    // =========================================================================
    // [1] RegisterAlarm ID — 倉儲區氣缸 (500-599) [Hold, Level2]
    // =========================================================================
    GC_ALARM_CYL_STO_UPCV_FEEDIN1       : DINT := 500;   // 上CV進料壓缸1
    GC_ALARM_CYL_STO_UPCV_FEEDIN2       : DINT := 501;   // 上CV進料壓缸2
    GC_ALARM_CYL_STO_UPCV_DIAMETER      : DINT := 502;   // 上CV量徑壓缸
    GC_ALARM_CYL_STO_UPCV_CAM1          : DINT := 503;   // 上CV相機壓缸1
    GC_ALARM_CYL_STO_UPCV_CAM2          : DINT := 504;   // 上CV相機壓缸2
    GC_ALARM_CYL_STO_UPCV_CAM3          : DINT := 505;   // 上CV相機壓缸3
    GC_ALARM_CYL_STO_UPCV_CAM4          : DINT := 506;   // 上CV相機壓缸4
    GC_ALARM_CYL_STO_UPCV_BLOCK1        : DINT := 507;   // 上CV擋塊1
    GC_ALARM_CYL_STO_UPCV_BLOCK2        : DINT := 508;   // 上CV擋塊2
    GC_ALARM_CYL_STO_UPCV_BLOCK3        : DINT := 509;   // 上CV擋塊3
    GC_ALARM_CYL_STO_UPCV_DIA_HORIZ     : DINT := 510;   // 上CV量徑水平
    GC_ALARM_CYL_STO_UPCV_DIA_VERT      : DINT := 511;   // 上CV量徑垂直
    GC_ALARM_CYL_STO_UPCV_DIA_CLAMP     : DINT := 512;   // 上CV量徑夾
    GC_ALARM_CYL_STO_STACK_PUSH         : DINT := 513;   // 疊盒推缸
    GC_ALARM_CYL_STO_LOWCV_PRESS1       : DINT := 514;   // 下CV壓缸1
    GC_ALARM_CYL_STO_LOWCV_PRESS2       : DINT := 515;   // 下CV壓缸2
    GC_ALARM_CYL_STO_LOWCV_PRESS3       : DINT := 516;   // 下CV壓缸3
    GC_ALARM_CYL_STO_LOWCV_PRESS4       : DINT := 517;   // 下CV壓缸4
    GC_ALARM_CYL_STO_LOWCV_BLOCK1       : DINT := 518;   // 下CV擋塊1
    GC_ALARM_CYL_STO_LOWCV_BLOCK2       : DINT := 519;   // 下CV擋塊2
    GC_ALARM_CYL_STO_SAME_BLOCK3        : DINT := 520;   // 同徑CV擋塊3
    GC_ALARM_CYL_STO_SHIP_BUFFER        : DINT := 521;   // 出貨緩衝壓缸
    // 522-599: 預留倉儲區氣缸擴充

    // =========================================================================
    // [1] RegisterAlarm ID — 配針區氣缸 (600-699) [Hold, Level2]
    // =========================================================================
    GC_ALARM_CYL_ALC_ROBOT_LCLAMP1      : DINT := 600;   // AllocateRobot 左夾1
    GC_ALARM_CYL_ALC_ROBOT_LCLAMP2      : DINT := 601;   // AllocateRobot 左夾2
    GC_ALARM_CYL_ALC_ROBOT_LVERT1       : DINT := 602;   // AllocateRobot 左升降1
    GC_ALARM_CYL_ALC_ROBOT_LVERT2       : DINT := 603;   // AllocateRobot 左升降2
    GC_ALARM_CYL_ALC_ROBOT_RCLAMP1      : DINT := 604;   // AllocateRobot 右夾1
    GC_ALARM_CYL_ALC_ROBOT_RCLAMP2      : DINT := 605;   // AllocateRobot 右夾2
    GC_ALARM_CYL_ALC_ROBOT_RVERT1       : DINT := 606;   // AllocateRobot 右升降1
    GC_ALARM_CYL_ALC_ROBOT_RVERT2       : DINT := 607;   // AllocateRobot 右升降2
    GC_ALARM_CYL_ALC_DIFF_BLOCK1        : DINT := 608;   // 異徑CV擋塊1
    GC_ALARM_CYL_ALC_RB_WORK_PRESS      : DINT := 609;   // 圓帶工作區壓缸
    GC_ALARM_CYL_ALC_RB_WORK_PLUG       : DINT := 610;   // 圓帶工作區插銷
    GC_ALARM_CYL_ALC_RB_CHARGE_PLUG     : DINT := 611;   // 圓帶充電區插銷
    GC_ALARM_CYL_ALC_RB_TRANS_PLUG      : DINT := 612;   // 圓帶傳送區插銷
    GC_ALARM_CYL_ALC_OUTROBOT_AVERT     : DINT := 613;   // OutRobot A側升降
    GC_ALARM_CYL_ALC_OUTROBOT_BVERT     : DINT := 614;   // OutRobot B側升降
    GC_ALARM_CYL_ALC_OUTROBOT_ACLAMP    : DINT := 615;   // OutRobot A側夾
    GC_ALARM_CYL_ALC_OUTROBOT_BCLAMP    : DINT := 616;   // OutRobot B側夾
    GC_ALARM_CYL_ALC_TRANS_CAMHORIZ     : DINT := 617;   // 傳送CV相機水平
    GC_ALARM_CYL_ALC_DIFF_PRESS2        : DINT := 618;   // 異徑CV壓缸2
    GC_ALARM_CYL_ALC_DIFF_PRESS1        : DINT := 619;   // 異徑CV壓缸1
    GC_ALARM_CYL_ALC_DIFF_BLOCK1_2      : DINT := 620;   // 異徑CV擋塊1 (重複)
    GC_ALARM_CYL_ALC_SAME_PRESS4        : DINT := 621;   // 同徑CV壓缸4
    GC_ALARM_CYL_ALC_SAME_PRESS3        : DINT := 622;   // 同徑CV壓缸3
    GC_ALARM_CYL_ALC_SAME_PRESS2        : DINT := 623;   // 同徑CV壓缸2
    GC_ALARM_CYL_ALC_SAME_PRESS1        : DINT := 624;   // 同徑CV壓缸1
    GC_ALARM_CYL_ALC_SAME_BLOCK2        : DINT := 625;   // 同徑CV擋塊2
    GC_ALARM_CYL_ALC_SAME_BLOCK1        : DINT := 626;   // 同徑CV擋塊1
    GC_ALARM_CYL_ALC_PULLOUT_APRESS1    : DINT := 627;   // 拔針CV A側壓缸1
    GC_ALARM_CYL_ALC_PULLOUT_APRESS2    : DINT := 628;   // 拔針CV A側壓缸2
    GC_ALARM_CYL_ALC_PULLOUT_ABLOCK     : DINT := 629;   // 拔針CV A側擋塊
    GC_ALARM_CYL_ALC_PULLOUT_BPRESS1    : DINT := 630;   // 拔針CV B側壓缸1
    GC_ALARM_CYL_ALC_PULLOUT_BPRESS2    : DINT := 631;   // 拔針CV B側壓缸2
    GC_ALARM_CYL_ALC_PULLOUT_BBLOCK     : DINT := 632;   // 拔針CV B側擋塊
    // 633-699: 預留配針區氣缸擴充

    // =========================================================================
    // [1] RegisterAlarm ID — 伺服軸 (800-899) [Abort, Level6]
    // =========================================================================
    GC_ALARM_AXIS_TURNTABLE              : DINT := 800;   // [Abort] 轉盤軸錯誤
    GC_ALARM_AXIS_ROUNDBELT              : DINT := 801;   // [Abort] 圓帶軸錯誤
    GC_ALARM_AXIS_ALLOCATE_X             : DINT := 802;   // [Abort] 配針X軸錯誤
    GC_ALARM_AXIS_ALLOCATE_Y             : DINT := 803;   // [Abort] 配針Y軸錯誤
    GC_ALARM_AXIS_OUTROBOT_X             : DINT := 804;   // [Abort] OutRobot X軸錯誤
    GC_ALARM_AXIS_OUTROBOT_Y             : DINT := 805;   // [Abort] OutRobot Y軸錯誤
    GC_ALARM_AXIS_RACKMOTOR              : DINT := 806;   // [Abort] RackMotor軸錯誤
    // 807-899: 預留伺服軸擴充
	
	GC_ALARM_MODBUSRTU					: DINT	:= 850;	  // 光電板 MODBUS (實際用 +1 ~ +4) 

    // =========================================================================
    // [1] RegisterAlarm ID — 安全門 (900-999) [Hold, Level2]
    // =========================================================================
    GC_ALARM_SAFE_DOOR_BASE              : DINT := 900;   // 安全門基底 (實際用 +1 ~ +16)
    // 917-999: 預留安全相關擴充

    // =========================================================================
    // [2] FB 內部錯誤碼 — 通用 (A=0, OO=00 一般)
    // =========================================================================
    GC_ERR_NONE                          : INT := 0;       // 無錯誤
    GC_ERR_TIMEOUT                       : INT := 1;       // 逾時 [Hold]
    GC_ERR_POSITION_INVALID              : INT := 3;       // 位置資料無效 [Hold]
    GC_ERR_INDEX_INVALID                 : INT := 10;      // 索引無效 [Hold]
    GC_ERR_WRONG_COMMAND                 : INT := 11;      // 錯誤指令 [Hold]
    GC_ERR_ROBOT_NUMBER_INVALID          : INT := 12;      // 機器人編號無效 [Hold]

    // -- 通用 氣缸 (A=0, OO=01) --
    GC_ERR_CYLINDER_NOT_READY            : INT := 102;     // 氣缸未就緒 [Hold]

    // -- 通用 馬達 (A=0, OO=02) --
    GC_ERR_MOTOR_NOT_READY               : INT := 202;     // 馬達未就緒 [Hold]

    // -- 通用 伺服軸 (A=0, OO=03) --
    GC_ERR_AXIS_NOT_READY                : INT := 302;     // 軸未就緒 [Hold]
    GC_ERR_AXIS_ERROR                    : INT := 310;     // 軸錯誤 [Abort]
    GC_ERR_AXIS_POSITION_ERROR           : INT := 305;     // 軸位置錯誤 [Hold]
    GC_ERR_AXIS_SAFETY_CALL_ERROR        : INT := 311;     // 呼叫軸安全檢查錯誤 [Abort]
    GC_ERR_AXIS_SAFETY_CHECK_ERROR       : INT := 312;     // 軸安全檢查錯誤 [Abort]
    GC_ERR_AXIS_OUTROBOT_X_ERROR        : INT := 313;     // OutRobot X軸錯誤 [Abort]
    GC_ERR_AXIS_OUTROBOT_Y_ERROR        : INT := 314;     // OutRobot Y軸錯誤 [Abort]
    GC_ERR_AXIS_ALLOCATE_X_ERROR        : INT := 315;     // 配針X軸錯誤 [Abort]
    GC_ERR_AXIS_ALLOCATE_Y_ERROR        : INT := 316;     // 配針Y軸錯誤 [Abort]
    GC_ERR_AXIS_ROUNDBELT_ERROR         : INT := 317;     // 圓帶軸錯誤 [Abort]
    GC_ERR_AXIS_TURNTABLE_ERROR         : INT := 318;     // 轉盤軸錯誤 [Abort]
    GC_ERR_RACKMOTOR_BTN_BLINK          : INT := 319;     // RackMotor按鈕閃爍 [Hold]
    GC_ERR_AXIS_X_NOT_READY             : INT := 320;     // X軸未就緒 [Hold]
    GC_ERR_AXIS_Y_NOT_READY             : INT := 321;     // Y軸未就緒 [Hold]

    // -- 通用 機器人 (A=0, OO=04) --
    GC_ERR_ROBOT_CANNOT_HOME             : INT := 410;     // 機器人無法回原點 [Abort]
    GC_ERR_ROBOT_REBOOT_TIMEOUT          : INT := 411;     // 機器人重啟逾時 [Abort]
    GC_ERR_ROBOT_CMD_NOT_BUSY            : INT := 412;     // 機器人指令未接受 [Hold]
    GC_ERR_ROBOT_CMD_TIMEOUT             : INT := 413;     // 機器人指令完成逾時 [Abort]
    GC_ERR_ROBOT_HOMING_ERROR            : INT := 414;     // 機器人回原點錯誤+訊息 [Abort]

    // =========================================================================
    // [2] FB 內部錯誤碼 — 倉儲區專用 (A=1)
    // =========================================================================
    GC_ERR_STO_ROBOT_FEEDOUT_NOT_BUSY    : INT := 10412;   // 倉儲機器人 FeedOut 未接受 [Hold]
    GC_ERR_STO_ROBOT_FEEDOUT_TIMEOUT     : INT := 10413;   // 倉儲機器人 FeedOut 逾時 [Abort]
    GC_ERR_STO_SERVICE_OCCUPIED          : INT := 10006;   // 倉儲服務佔用中 [Hold]

    // -- 倉儲區 下CV輸送帶 (A=1, OO=05/01) --
    GC_ERR_STO_LOWCV_BLOCK1_ERROR       : INT := 10110;   // 下CV擋塊1錯誤 [Hold]
    GC_ERR_STO_LOWCV_BLOCK2_ERROR       : INT := 10111;   // 下CV擋塊2錯誤 [Hold]
    GC_ERR_STO_LOWCV_PRESS1_ERROR       : INT := 10112;   // 下CV壓缸1錯誤 [Hold]
    GC_ERR_STO_LOWCV_PRESS2_ERROR       : INT := 10113;   // 下CV壓缸2錯誤 [Hold]
    GC_ERR_STO_LOWCV_PRESS3_ERROR       : INT := 10114;   // 下CV壓缸3錯誤 [Hold]
    GC_ERR_STO_LOWCV_PRESS4_ERROR       : INT := 10115;   // 下CV壓缸4錯誤 [Hold]
    GC_ERR_STO_LOWCV_BOX_TIMEOUT        : INT := 10501;   // 下CV盒子到位逾時 [Hold]
    GC_ERR_STO_LOWCV_CYL_ERROR          : INT := 10116;   // 下CV氣缸錯誤 (CyclicAction) [Hold]
    GC_ERR_STO_LOWCV_MOTOR_ERROR        : INT := 10201;   // 下CV馬達錯誤 (CyclicAction) [Hold]

    // =========================================================================
    // [2] FB 內部錯誤碼 — 配針區專用 (A=2)
    // =========================================================================
    GC_ERR_ALC_RB_NOT_READY              : INT := 20602;   // 圓帶軸未就緒 [Hold]
    GC_ERR_ALC_RB_CYLINDER_ERROR         : INT := 20102;   // 圓帶氣缸錯誤 [Hold]
    GC_ERR_ALC_RB_AXIS_ERROR             : INT := 20610;   // 圓帶軸錯誤 [Abort]
    GC_ERR_ALC_RB_CHARGE_PLUG_ERROR      : INT := 20111;   // 充電區插銷錯誤 [Hold]
    GC_ERR_ALC_RB_TRANSMITCV_PLUG_ERROR  : INT := 20511;   // 傳送帶插銷錯誤 [Hold]
    GC_ERR_ALC_RB_WORKZONE_PLUG_ERROR    : INT := 20112;   // 工作區插銷錯誤 [Hold]
    GC_ERR_ALC_RB_WORKZONE_PRESS_ERROR   : INT := 20113;   // 工作區壓缸錯誤 [Hold]
    GC_ERR_ALC_SERVO_ERROR               : INT := 20310;   // 配針伺服軸錯誤 [Abort]

    // -- 配針區 轉盤 (A=2, OO=07) --
    GC_ERR_ALC_TT_TARGET_INVALID        : INT := 20703;   // 轉盤目標無效 [Hold]
    GC_ERR_ALC_TT_AXIS_NOT_READY        : INT := 20702;   // 轉盤軸未就緒 [Hold]
    GC_ERR_ALC_TT_AXIS_ERROR            : INT := 20710;   // 轉盤軸錯誤 [Abort]
    GC_ERR_ALC_TT_CYLINDER_NOT_READY    : INT := 20701;   // 轉盤氣缸未就緒 [Hold]
    GC_ERR_ALC_TT_PRESS_ERROR           : INT := 20711;   // 轉盤壓缸錯誤 [Hold]

    // -- 配針區 同徑CV相機 (A=2) --
    GC_ERR_ALC_SAMECV_BLOCK1_ERROR      : INT := 20120;   // 同徑CV Block1錯誤 [Hold]
    GC_ERR_ALC_SAMECV_BLOCK2_ERROR      : INT := 20121;   // 同徑CV Block2錯誤 [Hold]
    GC_ERR_ALC_SAMECV_PRESS1_ERROR      : INT := 20122;   // 同徑CV Press1錯誤 [Hold]
    GC_ERR_ALC_SAMECV_PRESS2_ERROR      : INT := 20123;   // 同徑CV Press2錯誤 [Hold]
    GC_ERR_ALC_SAMECV_CAMHORIZ_ERROR    : INT := 20124;   // 同徑CV CameraHoriz錯誤 [Hold]
    GC_ERR_ALC_SAMECV_BOX_NOT_ARRIVED   : INT := 20515;   // 同徑CV 盒子未到逾時 [Hold]
    GC_ERR_ALC_SAMECV_CYL_TIMEOUT       : INT := 20125;   // 同徑CV 氣缸逾時 [Hold]
    GC_ERR_ALC_SAMECV_CAMERA_TIMEOUT    : INT := 20516;   // 同徑CV 拍照逾時 [Abort]
    GC_ERR_ALC_SAMECV_BOX_CROSS_TIMEOUT : INT := 20517;   // 同徑CV 盒子通過逾時 [Hold]
    GC_ERR_ALC_SAMECV_FULL              : INT := 20518;   // 同徑CV 滿載 [Hold]
    GC_ERR_ALC_SAMECV_MOTOR_ERROR       : INT := 20225;   // 同徑CV 馬達錯誤 [Hold]

    // -- 配針區 異徑CV相機 (A=2) --
    GC_ERR_ALC_DIFFCV_BLOCK1_ERROR      : INT := 20130;   // 異徑CV Block1錯誤 [Hold]
    GC_ERR_ALC_DIFFCV_PRESS1_ERROR      : INT := 20131;   // 異徑CV Press1錯誤 [Hold]
    GC_ERR_ALC_DIFFCV_CAMHORIZ_ERROR    : INT := 20132;   // 異徑CV CamaraHoriz錯誤 [Hold]
    GC_ERR_ALC_DIFFCV_NOT_READY         : INT := 20519;   // 異徑CV 未就緒 [Hold]
    GC_ERR_ALC_DIFFCV_CYL_TIMEOUT       : INT := 20133;   // 異徑CV 氣缸逾時 [Hold]
    GC_ERR_ALC_DIFFCV_BOX_NOT_ARRIVED   : INT := 20520;   // 異徑CV 盒子未到逾時 [Hold]
    GC_ERR_ALC_DIFFCV_CYL_MOTOR_TIMEOUT : INT := 20134;   // 異徑CV 馬達/氣缸逾時 [Hold]
    GC_ERR_ALC_DIFFCV_CAMERA_TIMEOUT    : INT := 20521;   // 異徑CV 拍照逾時 [Abort]
    GC_ERR_ALC_DIFFCV_BOX_CROSS_TIMEOUT : INT := 20522;   // 異徑CV 盒子通過逾時 [Hold]
    GC_ERR_ALC_DIFFCV_FULL              : INT := 20523;   // 異徑CV 滿載 [Hold]
    GC_ERR_ALC_DIFFCV_MOTOR_ERROR       : INT := 20226;   // 異徑CV 馬達錯誤 [Hold]

    // -- 配針區 逆向拍照批次入料 (A=2) --
    GC_ERR_ALC_REVBATCH_PICKUP_TIMEOUT  : INT := 20530;   // 逆向批次 小手臂取放盒逾時 [Hold]
    GC_ERR_ALC_REVBATCH_BIGARM_TIMEOUT  : INT := 20531;   // 逆向批次 大手臂搬運逾時 [Hold]
    GC_ERR_ALC_REVBATCH_CONVEYOR_FULL   : INT := 20532;   // 逆向批次 軌道滿載 [Hold]
    GC_ERR_ALC_REVBATCH_CONFIG_TIMEOUT  : INT := 20533;   // 逆向批次 等待C#配置逾時 [Hold]
    GC_ERR_ALC_REVBATCH_CAMERA_TIMEOUT  : INT := 20534;   // 逆向批次 拍照逾時 [Hold]

    // =========================================================================
    // [2] FB 內部錯誤碼 — 出貨區專用 (A=3)
    // =========================================================================
    GC_ERR_SHP_ROBOT_FEEDOUT_NOT_BUSY    : INT := 30412;   // 出貨機器人 FeedOut 未接受 [Hold]
    GC_ERR_SHP_ROBOT_FEEDOUT_TIMEOUT     : INT := 30413;   // 出貨機器人 FeedOut 逾時 [Abort]
    GC_ERR_SHP_SERVICE_OCCUPIED          : INT := 30006;   // 出貨服務佔用中 [Hold]
    GC_ERR_SHP_ROBOT_REBOOT_TIMEOUT      : INT := 30411;   // 出貨機器人重啟逾時 [Abort]

    // -- 出貨區 雷射/傳送帶 (A=3) --
    GC_ERR_SHP_LASER_ERROR              : INT := 30910;   // 雷射機台錯誤 [Hold]
    GC_ERR_SHP_TRANSCV_NOT_IN_POS       : INT := 30511;   // 傳送帶未在目標位置 [Hold]

    // =========================================================================
    // [3] 服務唯一識別碼 — UniqueErrorCode (INT)
    //     各 Service FB 的 ErrorID，用於錯誤追蹤定位
    // =========================================================================
    // -- 倉儲區機器人服務 --
    GC_SVCID_STO_ROBOT_ABS_MOVE         : INT := 2200;   // 倉儲機器人絕對移動
    GC_SVCID_STO_REGION_ALLOC_CV        : INT := 2210;   // 區域移動-配針輸送帶
    GC_SVCID_STO_REGION_ROUNDBELT       : INT := 2220;   // 區域移動-圓帶
    GC_SVCID_STO_REGION_PULLOUT_CV      : INT := 2230;   // 區域移動-拔針輸送帶
    GC_SVCID_STO_REGION_FEEDIN_CV       : INT := 2240;   // 區域移動-進料輸送帶
    GC_SVCID_STO_WAREHOUSE_ROBOT        : INT := 2400;   // 倉儲機器人移動
    GC_SVCID_STO_ADD_BOXES              : INT := 2700;   // 加盒服務
    GC_SVCID_STO_UPPER_FEEDIN_CV        : INT := 2710;   // 上層進料輸送帶
    GC_SVCID_STO_BOX_SUPPLY             : INT := 2800;   // 供盒控制

    // -- 配針區服務 --
    GC_SVCID_ALC_PULLOUT_CV             : INT := 2750;   // 拔針輸送帶
    GC_SVCID_ALC_BATCH_SIMPLE           : INT := 112;    // 批次配針(簡易模式)
    GC_SVCID_ALC_BATCH_FULL             : INT := 108;    // 批次配針(完整模式)

    // -- 出貨區機器人服務 --
    GC_SVCID_SHP_ROBOT                  : INT := 2250;   // 出貨機器人


    // =========================================================================
    // [3] 中央化狀態訊息常數
    // =========================================================================
    GC_MSG_0001                      : STRING := 'Action Robot timeout';
    GC_MSG_0002: STRING := 'BlockBox1 MoveForward or BlockBox2 MoveBackward or DiameterMeasurementPressBox MoveBackward timeout';
    GC_MSG_0003           : STRING := 'Block 1 cylinder inrearPosition';
    GC_MSG_0004           : STRING := 'Block 2 cylinder inrearPosition';
    GC_MSG_0005             : STRING := 'Block box on conveyor timeout';
    GC_MSG_0006                     : STRING := 'box1 diameter timeout';
    GC_MSG_0007: STRING := 'Box not at Input.bUpCV_Block2Detect_Sensor';
    GC_MSG_0008                      : STRING := 'Box not On Turntable';
    GC_MSG_0009                      : STRING := 'Box Not on Turntable';
    GC_MSG_0010                                 : STRING := 'Box on A1';
    GC_MSG_0011                                 : STRING := 'Box on A2';
    GC_MSG_0012                          : STRING := 'Box On Turntable';
    GC_MSG_0013                           : STRING := 'Box still on A1';
    GC_MSG_0014                           : STRING := 'Box still on A2';
    GC_MSG_0015                     : STRING := 'Box still on conveyor';
    GC_MSG_0016                    : STRING := 'Box still on Turntable';
    GC_MSG_0017       : STRING := 'Check FirstBoxCamaraDone info retry';
    GC_MSG_0018                        : STRING := 'ClampA Robot Error';
    GC_MSG_0019                    : STRING := 'Clamp A Feedin timeout';
    GC_MSG_0020                    : STRING := 'Clamp A reload timeout';
    GC_MSG_0021                     : STRING := 'Clamp A robot timeout';
    GC_MSG_0022                    : STRING := 'Clamp B Feedin timeout';
    GC_MSG_0023                    : STRING := 'Clamp B reload timeout';
    GC_MSG_0024                     : STRING := 'Clamp B Robot timeout';
    GC_MSG_0025                   : STRING := 'Clip pick close timeout';
    GC_MSG_0026                   : STRING := 'clip pick close timeout';
    GC_MSG_0027                   : STRING := 'clip place open timeout';
    GC_MSG_0028                   : STRING := 'Clip place open timeout';
    GC_MSG_0029: STRING := 'Command error : Clamp A target layer out of range.';
    GC_MSG_0030: STRING := 'Command error : Clamp A target slide out of range';
    GC_MSG_0031: STRING := 'Command error : Clamp B target layer out of range.';
    GC_MSG_0032: STRING := 'Command error : Clamp B target slide out of range';
    GC_MSG_0033                   : STRING := 'Controller report error';
    GC_MSG_0034: STRING := 'Conveyor not ready , please remove boxes in front';
    GC_MSG_0035: STRING := 'Cylinder.List.fbUpCV_Block2 MoveForward timeout';
    GC_MSG_0036       : STRING := 'Cylinder.List.fbUpCV_Block3 timeout';
    GC_MSG_0037: STRING := 'Cylinder.List.fbUpCV_CamaraPress1.M_MoveForward timeout';
    GC_MSG_0038: STRING := 'Cylinder.List.fbUpCV_CamaraPress1 or Cylinder.List.fbUpCV_Block3 InRearPosition timeout';
    GC_MSG_0039: STRING := 'Cylinder.List.fbUpCV_DiameterClamp M_Extend Timeout';
    GC_MSG_0040: STRING := 'Cylinder.List.fbUpCV_DiameterClamp M_Retract Timeout';
    GC_MSG_0041: STRING := 'Cylinder.List.fbUpCV_DiameterHoriz M_Extend Timeout';
    GC_MSG_0042: STRING := 'Cylinder.List.fbUpCV_DiameterHoriz M_Retract Timeout';
    GC_MSG_0043: STRING := 'Cylinder.List.fbUpCV_DiameterPress MoveForward timeout';
    GC_MSG_0044: STRING := 'Cylinder.List.fbUpCV_DiameterVert MoveForward Timeout';
    GC_MSG_0045: STRING := 'Cylinder.List.fbUpCV_DiameterVert M_Extend Timeout';
    GC_MSG_0046: STRING := 'Cylinder.List.fbUpCV_DiameterVert M_Retract Timeout';
    GC_MSG_0047: STRING := 'Cylinder.List.fbUpCV_FeedInPress1 or Cylinder.List.fbUpCV_FeedInPress2 MoveForward timeout';
    GC_MSG_0048                : STRING := 'Cylinder pick down timeout';
    GC_MSG_0049                  : STRING := 'Cylinder pick up timeout';
    GC_MSG_0050                  : STRING := 'cylinder pick up timeout';
    GC_MSG_0051               : STRING := 'Cylinder place down timeout';
    GC_MSG_0052                 : STRING := 'Cylinder place up timeout';
    GC_MSG_0053                 : STRING := 'cylinder place up timeout';
    GC_MSG_0054       : STRING := 'C# DiameterMovement Pickdone timeout';
    GC_MSG_0055   : STRING := 'C# FirstBoxCameraDiameterRequest timeout';
    GC_MSG_0056              : STRING := 'C# FirstBoxCameraDone timeout';
    GC_MSG_0057     : STRING := 'C# SecondBoxCameraDiameterDone timeout';
    GC_MSG_0058                          : STRING := 'Data not correct';
    GC_MSG_0059  : STRING := 'Destination: Left TransCV not in position';
    GC_MSG_0060 : STRING := 'Destination: Right TransCV not in position';
    GC_MSG_0061                    : STRING := 'Empty conveyor timeout';
    GC_MSG_0062                    : STRING := 'Empty Conveyor timeout';
    GC_MSG_0063                       : STRING := 'Empty Robot timeout';
    GC_MSG_0064           : STRING := '_fbDiameterMovement Done timeout';
    GC_MSG_0065        : STRING := 'FeedInBox1Detecting not have a box';
    GC_MSG_0066: STRING := 'FeedInPressBox1Cylinder or FeedInPressBox2Cylinder or ReadCodePressBox2Cylinder MoveBackward timeout';
    GC_MSG_0067                            : STRING := 'Feed box error';
    GC_MSG_0068                          : STRING := 'Feed box timeout';
    GC_MSG_0069                          : STRING := 'Feed Box timeout';
    GC_MSG_0070                : STRING := 'First box diameter timeout';
    GC_MSG_0071: STRING := 'First box still at Input.bUpCV_Block2Detect_Sensor';
    GC_MSG_0072                  : STRING := 'FROM: Reset Robot timeout';
    GC_MSG_0073                 : STRING := 'FROM: Robot action timeout';
    GC_MSG_0074                : STRING := 'Get command, clamp have box';
    GC_MSG_0075                : STRING := 'Get command , clamp have box';
    GC_MSG_0076: STRING := 'Input.bUpCV_Block2Detect_Sensor not have box';
    GC_MSG_0077: STRING := 'Input.bUpCV_Block3Detect_Sensor first box leave timeout';
    GC_MSG_0078        : STRING := 'Lowerconveyor Reverse Stop timeout';
    GC_MSG_0079             : STRING := 'Lowerconveyor Reverse timeout';
    GC_MSG_0080                   : STRING := 'Modbus connection error';
    GC_MSG_0081                      : STRING := 'Move box out timeout';
    GC_MSG_0082    : STRING := 'Move Robot to picking position timeout';
    GC_MSG_0083    : STRING := 'Move robot to picking position timeout';
    GC_MSG_0084    : STRING := 'Move robot to placing position timeout';
    GC_MSG_0085   : STRING := 'Move Robot to placing position time out';
    GC_MSG_0086                              : STRING := 'No Box on A1';
    GC_MSG_0087                              : STRING := 'No Box on A2';
    GC_MSG_0088                        : STRING := 'No Box on conveyor';
    GC_MSG_0089                                  : STRING := 'No Error';
    GC_MSG_0090                                  : STRING := 'No error';
    GC_MSG_0091                                  : STRING := 'no error';
    GC_MSG_0092                         : STRING := 'no error , retrying';
    GC_MSG_0093    : STRING := 'Pick Box ClampA from RoundBelt timeout';
    GC_MSG_0094    : STRING := 'Pick Box ClampB from RoundBelt timeout';
    GC_MSG_0095           : STRING := 'Pick Box from RoundBelt timeout';
    GC_MSG_0096                          : STRING := 'Pick Box timeout';
    GC_MSG_0097                         : STRING := 'Place Box timeout';
    GC_MSG_0098            : STRING := 'Place Box to WareHouse timeout';
    GC_MSG_0099          : STRING := 'Place command , clamp not have box';
    GC_MSG_0100          : STRING := 'Place command, clamp not have box';
    GC_MSG_0101    : STRING := 'Prepare Cylinder clear command timeout';
    GC_MSG_0102: STRING := 'PullOutConveyorA FeedIn full box ,please remove box';
    GC_MSG_0103: STRING := 'PullOutConveyorA FeedOut full box ,please remove';
    GC_MSG_0104   : STRING := 'PullOutConveyorA full box ,please remove';
    GC_MSG_0105: STRING := 'PullOutConveyorA none box ,please refill box';
    GC_MSG_0106: STRING := 'PullOutConveyorB FeedIn full box ,please remove box';
    GC_MSG_0107: STRING := 'PullOutConveyorB FeedOut full box ,please remove';
    GC_MSG_0108   : STRING := 'PullOutConveyorB full box ,please remove';
    GC_MSG_0109                  : STRING := 'Rackmotor moving timeout';
    GC_MSG_0110              : STRING := 'RackPusher move back timeout';
    GC_MSG_0111           : STRING := 'RackPusher move forward timeout';
    GC_MSG_0112     : STRING := 'Rack occupied by user Push FeedButton';
    GC_MSG_0113                       : STRING := 'Reset Robot timeout';
    GC_MSG_0114: STRING := 'Robot A Clamp Get Box , Clamp has box or Clamp not Open';
    GC_MSG_0115: STRING := 'Robot A Clamp Place Box , Clamp not has box or Clamp Open';
    GC_MSG_0116: STRING := 'Robot both Clamp Get Box , Clamp has box or Clamp not has open';
    GC_MSG_0117: STRING := 'Robot both Clamp Place Box , Clamp not has box or Clamp has open';
    GC_MSG_0118: STRING := 'Robot B Clamp Get Box , Clamp has box or Clamp not has open';
    GC_MSG_0119: STRING := 'Robot B Clamp Place Box , Clamp not has box or Clamp has open';
    GC_MSG_0120: STRING := 'Robot do Only A Clamp Get Box , Clamp has box or Clamp not Open';
    GC_MSG_0121: STRING := 'Robot do Only A Clamp Place Box , Clamp not has box or Clamp Open';
    GC_MSG_0122: STRING := 'Robot do Only B Clamp Get Box , Clamp has box or Clamp not has open';
    GC_MSG_0123: STRING := 'Robot do Only B Clamp Place Box , Clamp not has box or Clamp has open';
    GC_MSG_0124                               : STRING := 'Robot Error';
    GC_MSG_0125                           : STRING := 'Robot Has Fault';
    GC_MSG_0126                        : STRING := 'Robot move timeout';
    GC_MSG_0127                        : STRING := 'Robot Move timeout';
    GC_MSG_0128    : STRING := 'Robot move to picking position timeout';
    GC_MSG_0129    : STRING := 'robot move to placing position timeout';
    GC_MSG_0130                           : STRING := 'RoundBelt Error';
    GC_MSG_0131: STRING := 'Second box feedin to read code camera pos timeout';
    GC_MSG_0132       : STRING := 'Source: Left TransCV not in position';
    GC_MSG_0133      : STRING := 'Source: Right TransCV not in position';
    GC_MSG_0134                         : STRING := 'Station get Error';
    GC_MSG_0135                     : STRING := 'Stop Conveyor timeout';
    GC_MSG_0136                     : STRING := 'Stop conveyor timeout';
    GC_MSG_0137                        : STRING := 'Stop Robot timeout';
    GC_MSG_0138: STRING := 'There is a box on Input.bUpCV_Block1Detect_Sensor';
    GC_MSG_0139                    : STRING := 'TO: Reset Robot timeout';
    GC_MSG_0140                   : STRING := 'TO: Robot action timeout';
    GC_MSG_0141                 : STRING := 'Use bothClamp robot Error';
    GC_MSG_0142            : STRING := 'Use ClampA Command Robot Error';
    GC_MSG_0143            : STRING := 'Use ClampB Command Robot Error';
    GC_MSG_0144                    : STRING := 'Use ClampB Robot Error';
    GC_MSG_0145         : STRING := 'wait Box Arrived TransCV time out';
    GC_MSG_0146                             : STRING := 'Wrong command';
    GC_MSG_0147            : STRING := 'Wrong command ,Area_A not allow';
    GC_MSG_0148  : STRING := 'Wrong command ,Area A not match to Area B';
    GC_MSG_0149            : STRING := 'Wrong command ,Area_B not allow';
    GC_MSG_0150            : STRING := 'Wrong command ,Both Area are 99';
    GC_MSG_0151    : STRING := 'Wrong command , Both warehouses selected';
    GC_MSG_0152: STRING := 'Wrong command, Buffer Position must be 1-55';
    GC_MSG_0153: STRING := 'Wrong command ,Can Not Get box from FeedOut conveyor';
    GC_MSG_0154: STRING := 'Wrong command ,Can Not Put box to FeedIn conveyor';
    GC_MSG_0155   : STRING := 'Wrong command, check the command setting';
    GC_MSG_0156             : STRING := 'Wrong command ,Clamp B has box';
    GC_MSG_0157     : STRING := 'Wrong command: Clip A target not allow';
    GC_MSG_0158     : STRING := 'Wrong command: Clip B target not allow';
    GC_MSG_0159      : STRING := 'Wrong command ,GetA not match to GetB';
    GC_MSG_0160: STRING := 'Wrong command, Left/Right Position must be 1-40';
    GC_MSG_0161  : STRING := 'Wrong command, no clamp has Work behavior';
    GC_MSG_0162       : STRING := 'Wrong command , No warehouse selected';
    GC_MSG_0163      : STRING := 'Wrong command ,Position A Not allowed';
    GC_MSG_0164        : STRING := 'Wrong command ,Position A Not allow';
    GC_MSG_0165      : STRING := 'Wrong command ,Position B Not allowed';
    GC_MSG_0166        : STRING := 'Wrong command ,Position B Not allow';
    GC_MSG_0167     : STRING := 'Wrong command ,TransCV not In Position';
    GC_MSG_0168: STRING := 'Wrong command, TransmitCVEnd Position must be 1-2';
    GC_MSG_0169                : STRING := 'Wrong command, unknown Area';
    GC_MSG_0170  : STRING := 'Wrong Command ,UseA and UseB both not use';
    GC_MSG_0171   : STRING := 'Wrong command ,use Clamp Command invaild';
    GC_MSG_0172   : STRING := 'Pick pos lost: OutRobot XY drifted before clip down';
    GC_MSG_0173   : STRING := 'Place pos lost: OutRobot XY drifted before clip down';
    GC_MSG_0174   : STRING := 'TurnTable interlock: must not move while clip down';
    GC_MSG_0175   : STRING := 'TurnTable angle invalid: must be 0/90/180/270/360';

    // === MachineControl central alarms (0176-0203) ===
    // EStop / AirPressure
    GC_MSG_0176   : STRING := 'Allocate Estop has trig';
    GC_MSG_0177   : STRING := 'Storage Estop has trig';
    GC_MSG_0178   : STRING := 'Storage robot Estop has trig';
    GC_MSG_0179   : STRING := 'Shipping robot Estop has trig';
    GC_MSG_0180   : STRING := 'Low AirPressure ';
    // Axis errors
    GC_MSG_0181   : STRING := 'TurnTable axis has Error';
    GC_MSG_0182   : STRING := 'Roundbelt axis has Error';
    GC_MSG_0183   : STRING := 'Allocate_X axis has Error';
    GC_MSG_0184   : STRING := 'Allocate_Y axis has Error';
    GC_MSG_0185   : STRING := 'OutRobot_X axis has Error';
    GC_MSG_0186   : STRING := 'OutRobot_Y axis has Error';
    GC_MSG_0187   : STRING := 'RackMotor axis has Error';
    // Safe doors (1-14, preserving existing typos/spacing)
    GC_MSG_0188   : STRING := 'Safe door1  Opened';
    GC_MSG_0189   : STRING := 'Safe door2  Opened';
    GC_MSG_0190   : STRING := 'Safe door3  Opened';
    GC_MSG_0191   : STRING := 'Safe door4  Opened';
    GC_MSG_0192   : STRING := 'Safe door5  Opened';
    GC_MSG_0193   : STRING := 'Safe door6  Opened';
    GC_MSG_0194   : STRING := 'Safe door7  Opened';
    GC_MSG_0195   : STRING := 'Safe door8  Opened';
    GC_MSG_0196   : STRING := 'Safe door9  Opened';
    GC_MSG_0197   : STRING := 'Safe door10  Opened';
    GC_MSG_0198   : STRING := 'Safe door11  Opened';
    GC_MSG_0199   : STRING := 'Safe doo12  Opened';
    GC_MSG_0200   : STRING := 'Safe doo13  Opened';
    GC_MSG_0201   : STRING := 'Safe door14  Opened';
    GC_MSG_0202   : STRING := 'Allocate_Electrical_Cabinet_SafetyDoor  Opened';
    GC_MSG_0203   : STRING := 'bShippingRobot_ElectricalCabinet_SafetyDoor  Opened';

    // === FanucRobot runtime status (0204-0221) ===
    GC_MSG_0204   : STRING := 'EStop has been trigged.';
    GC_MSG_0205   : STRING := 'Get but Has Sensor no Respond';
    GC_MSG_0206   : STRING := 'Get But Jaw Has';
    GC_MSG_0207   : STRING := 'illegal value in tool offset';
    GC_MSG_0208   : STRING := 'Jaw Sensor no Respond';
    GC_MSG_0209   : STRING := 'Laser detected';
    GC_MSG_0210   : STRING := 'Read All offset data failue';
    GC_MSG_0211   : STRING := 'Retry too many times, Need Robot Homing';
    GC_MSG_0212   : STRING := 'Robot Disconnect';
    GC_MSG_0213   : STRING := 'Robot has Battary alarm';
    GC_MSG_0214   : STRING := 'Robot has fatal alarm';
    GC_MSG_0215   : STRING := 'Robot in Halt State';
    GC_MSG_0216   : STRING := 'Robot Not in Home Pos, Home First';
    GC_MSG_0217   : STRING := 'RSR1 has error when RSR1 active.Restart Robot Power.';
    GC_MSG_0218   : STRING := 'RSR3 has error when RSR3 active.';
    GC_MSG_0219   : STRING := 'TP has got contol';
    GC_MSG_0220   : STRING := 'Upper data Overload';
    GC_MSG_0221   : STRING := 'Vision fault';

END_VAR

// ---- Library/10_Machine/18_HMI_Handshake/GVL_ADS.TcGVL
{attribute 'qualified_only'}
VAR_GLOBAL
	
//========單動一行程============
//    // one process use
    //配針單動資料結構
    AllocateMoveStructure : st_ads_AllocateMoveStructure;
	//拔針單動資料結構
    AllocateMoveStructure_Reverse : st_ads_AllocateMoveStructure;     
    //空盒手臂單動資料結構
    EmptyRobotToTurnTableMove : st_ads_OneAxisMoveWithPosition;
    //圓帶單動一行程
    AllocateCircleMove : st_AllocateCircleMoveStructure;
    //圓盤單動一行程
    TurnTableMove : st_ads_OneAxisMoveWithPosition;
//    //軸還原預設狀態
//    AxesControl : ARRAY[0..10] OF st_AxisControl;
    //機台還原預設狀態
    MachineReset : st_ads_MachineReset;
    //Empty
    RareFullBoxPush : st_ads_OutRobtToPlateMove;
	
	// Move Allocate robot to needling position
	AllocationRobotNeedlingMove : st_AllocateRobotNeedlingMove;

//==============自動模式=========================

    //AutoModeUse*-------自動模式圓帶單動
    AutoMode_AllocateCircleMove : st_AllocateCircleMoveStructure;
    //AutoModeUse*-------手臂倉儲位置移動
    AutoMode_RobotWarehouseMove : st_AutoSixAxisWarehouseParameter;
    //AutoModeUse*-------手臂絕對位置移動
    AutoMode_RobotAbsMove : st_AutoSixAxisAbsMoveParameter;
    //AutoModeUse*-------空盒取料移動
    AutoMode_EmptyBoxMove : st_AutoMode_ClampingBoxesJob;
    //AutoModeUse*-------圓盤移動
    AutoMode_TurnTableMove : st_ads_OneAxisMoveWithPosition;
    //AutoModeUse--------配針
    AutoMode_AllocateMove : st_AutoMode_AllocatingJob;
	 //AutoModeUse--------拔針
    AutoMode_AllocateMove_Reverse : st_AutoMode_AllocatingJob;
	//AutoModeUse--------配針batch mode
	AutoMode_AllocateBatchMode	:ST_AllocationJobBatchMode;
	//AutoModeUse--------拔針batch mode
	AutoMode_AllocateBatchMode_Reverse	:ST_AllocationJobBatchMode;
	//AutoModeSimpleAllocation_Batch
	AutoMode_SimpleAllocation_Batch		:ST_AllocationJobBatchMode;
    //AutoMdeUse---------散針放盒
    AutoMode_RareBoxMove : st_AutoMode_ClampingBoxesJob;
    //AutoMdeUse---------出貨放盒單動
    AutoMode_OutBoxMove : st_AutoMode_ClampingToPlate;
	//AutoMdeUse---------拔針放盒自動模式
    AutoMode_BoxMoveReverse : st_AutoMode_ClampingBoxesJob;
    //倉儲分選區移動,移動位置列表需延伸此陣列取得 WarehouseMovePosition :ARRAY[0..3] OF st_OneDirectionCore;
    AutoMode_WarehouseMove : st_ads_OneAxisMoveWithPosition;
    //AutoModeUse------手臂區域移動_FeedIn conveyor
	AutoMode_RobotRegionMove_FeedInConveyor		:ST_AutoMode_RobotRegionMove;
	//AutoModeUse------手臂區域移動_AllocatedConveyor
	AutoMode_RobotRegionMove_AllocatedConveyor		:ST_AutoMode_RobotRegionMove;
	//AutoModeUse------手臂區域移動_Pullout conveyor
	AutoMode_RobotRegionMove_PullOutConveyor		:ST_AutoMode_RobotRegionMove;
	//AutoModeUse------手臂區域移動_Buffer area
	AutoMode_RobotRegionMove_BufferArea		:ST_AutoMode_RobotRegionMove;
	//AutoModeUse------手臂區域移動_RoundBelt
	AutoMode_RobotRegionMove_RoundBelt		:ST_AutoMode_RobotRegionMove;
   //AutoMode MoveConveyorJob------定時移動輸送帶
    AutoMode_MoveConveyorJob : st_MoveConveyorJob;
	// Automode Feedin empty box with robot 
	AutoMode_FeedInEmptyBoxWithRobot : ST_AutoMode_FeedInEmptyBox; // Automode : Feedin empty box with robot from Warehouse and Pullout convenyor
	// Automode Reload RoundBelt box with robot
	AutoMode_ReloadRoundBeltBoxWithRobot : ST_AutoMode_ReloadRoundBeltBox; // Automode : Reload RoundBelt box with robot from warehouse
	// Automode FeedIn RoundBelt box to warehouse - 圓帶到倉儲		edited Gamin 2026/04/02 
	AutoMode_FeedInRoundBeltBoxToWareHouse : ST_AutoMode_FeedInToWareHouseBox; // Automode : Pick box from RoundBelt and place to WareHouse
	//AutoMode UpperFeedInConveyor
	AutoMode_UpperFeedInConveyor : ST_Auto_UpperFeedInConveyor;
	//AutoModeUse------倉儲馬達搭配手臂移動
    AutoMode_WarehouseMotoWithRobotMove : st_AutoSixAxisWarehouseParameter;
    //SimpleAllocate Autode-----簡易配針
	AutoMode_SimpleAllocate    : ST_AutoMode_SimpleAllocateHandShake; // AutoMode Simple Allocate
    AutoMode_PullOutConveyor   : ST_AutoPullOutConveyor; // AutoMode PullOut Conveyor
    //AutoModeUse----------錯誤通知  Host To PLC
    AutoMode_ErrorHandle : ST_Alarm;
    //Alarm report	----------錯誤通知 PLC to Host
    AlarmAllocation : ARRAY[0..999] OF ST_Alarm_Tmax;
	//AutoMode Use------ShippingGoodV2		20250304 Min
	AutoMode_AddBoxes	:ST_AutoAddsBoxes;
    //=================TwinCat Memory============
    //TwinCatMemory				:st_TwinCatMemory;
    //=================全局Home===================

    MachineHome          : st_RegionHome; // Machine all units home command
    StorageRegionHome    : st_RegionHome;
    AllocationRegionHome : st_RegionHome;
    FGARegionHome        : st_RegionHome;

    //===============手自動=======================
    StorageRegionMode : ST_Mode;
    AllocationRegion  : ST_Mode;
    FGARegionMode     : ST_Mode;
    MachineMode       : ST_Mode;
	
    // Operation Pannel Status
    OpPannel_Status : ST_OpPannelStatus; //PLC -> HMI
    OpPannel_Ctrl   : ST_OpPannelStatus; // HMI -> PLC

	//20250425 addon
	//Machine state
	MachineState : E_MachineState :=E_MachineState.Default;
	
	FanucRobot_General               : ST_FanucRobotGeneralCtrl;
	
	//AutoModeUse------倉儲小手臂ABS 移動
	AutoMode_ShippingRobot_Left            : ST_AutoMode_ShippingRobot_MoveAbs;
	//AutoModeUse------倉儲小手臂ABS 移動
	AutoMode_ShippingRobot_Right           : ST_AutoMode_ShippingRobot_MoveAbs;
	//AutoModeUse------倉儲小手臂ABS 移動
	AutoMode_ShippingRobot_TransmitCVEnd    : ST_AutoMode_ShippingRobot_MoveAbs;
	//AutoModeUse------同尺寸拍照
	AutoMode_SameSizeCVCamera				: ST_AutoMode_TransCVCamera;
	//AutoModeUse------同尺寸反向拍照
	AutoMode_SameSizeCVCamera_Reverse		: ST_AutoMode_TransCVCamera;
	//AutoModeUse------不同尺寸拍照
	AutoMode_DifferentCVCamera				: ST_AutoMode_TransCVCamera;
	//AutoModeUse------逆向拍照批次入料
	AutoMode_ReverseBatchPick				: ST_AutoMode_ReverseBatchPick;
	//AutoModeUse------同尺寸軌道回倉/NG
	AutoMode_ReverseBoxToWareHouse			: ST_AutoMode_ReverseBoxToWareHouse;
		
	//Shipping FeedOut TransCV with HansLaser handshake Service
	AutoMode_ShippingLeftSideTransCV		: ST_AutoMode_ShippingLeftSideTransCV;
	AutoMode_ShippingRightSideTransCV		: ST_AutoMode_ShippingRightSideTransCV;
	//AutoModeUse------倉儲內取放圓帶 (單筆)
	AutoMode_WareHouseInnerPickToRoundBelt		: ST_AutoMode_WareHouseInnerPickToRoundBelt;
	//AutoModeUse------倉儲內取放圓帶 (批次)
	AutoMode_WareHouseInnerPickToRoundBeltBatch	: ST_WareHouseInnerPickBatch;
	//AutoModeUse------圓帶回倉/PullOut (批次)
	AutoMode_FeedInRoundBeltBoxBatch			: ST_FeedInRBBatch;
	//Reboot Modbus devices
	RebootModbusDevices			: st_RebootModbusDevices;
	//AutoModeUse------- 出貨區緩衝區
	AutoMode_ShippingRobot_Buffer			: ST_AutoMode_ShippingRobot_MoveAbs;
	//AutoModeUse------- 出貨區拍照位置
	AutoMode_ShippingRobot_PhotoStandByPos	: ST_AutoMode_ShippingRobot_MoveAbs;
	//AutoModeUse------- 出貨區搬運 (合併)
	AutoMode_ShippingRobotTransfer			: ST_AutoMode_ShippingRobotTransfer;
	//AutoModeUse------- 出貨區小手臂鐵盤掃描
	AutoMode_ShippingPlateScan				: ST_ShippingPlateToConveyor;
	//AutoModeUse------- 手臂單獨回原點
	AutoMode_RobotSelfHoming				: ST_AutoMode_RobotSelfHoming;
	//BuzzCtrl 
	BuzzCtrl								: ST_BuzzCtrl;
	
END_VAR

// ---- Library/10_Machine/18_HMI_Handshake/GVL_HMI.TcGVL
{attribute 'qualified_only'}
VAR_GLOBAL
	OpMode : E_UnitMode; // Only Manual and Auto
    Allocated : ST_HMI_AllocateArea;
    Storage   : ST_HMI_StorageArea;
    Shipping  : ST_HMI_ShippingArea;
    IOMonitor : ST_HMI_IOMonitor;
    Setup     : ST_SetupPara;
    Status    : ST_HMI_MachineStatus;
END_VAR

// ---- Library/30_Simulation/GVL_SimMode.TcGVL
{attribute 'qualified_only'}
VAR_GLOBAL
    // TRUE = 數位孿生模擬模式；使用時在 DAS_CoreSys 傳入 MachineControl(EnableSimulation := GVL_SimMode.bSimMode)
    bSimMode : BOOL := FALSE;
END_VAR

// ---- POUs/ModbusRTU/ComModbusRTU.TcPOU
PROGRAM ComModbusRTU
VAR
	MB_EL6X22B_ControllerN				:	ARRAY[0..3] OF ModbusRtuMasterV2_KL6x22B;
	MBUnusedData_Read 					: 	ARRAY[0..3] OF ARRAY[0..7] OF BYTE;
	MBSensorError_Read 					: 	ARRAY[0..3] OF ARRAY[0..21] OF BYTE;
	nErrID_ControllerN					:	ARRAY[0..3] OF MODBUS_ERRORS;
	iReadMBAddr							:	ARRAY[0..3] OF WORD;
	bBusy_ControllerN					:	ARRAY[0..3] OF BOOL;
	bError_ControllerN					:	ARRAY[0..3] OF BOOL;
	fbComReset_ControllerN				:	ARRAY[0..3] OF ComReset;
	bComReset							:	ARRAY[0..3] OF BOOL;
	bComResetBusy							:	ARRAY[0..3] OF BOOL;
	bComResetError							:	ARRAY[0..3] OF BOOL;
	bStart								:	ARRAY[0..3] OF BOOL;
	
	actStart							:	ARRAY[0..3] OF ULINT;
	actEnd								:	ARRAY[0..3] OF ULINT;
	exeTime								:	ARRAY[0..3] OF ULINT;
	nSlave								:	BYTE;
	MBdata_Read_ControllerN	 AT %I*		: 	ARRAY[0..3] OF ARRAY[0..21] OF BYTE;
	bMasterError						:	ARRAY[0..3] OF BOOL;
	nStep								:	UINT;
	bModbusRTUError						:	BOOL;
	udiModbusRTUErrorID					:	UDINT;
	nAlias								:	UINT;
	bPassModBusMaster					:	ARRAY[0..3] OF BOOL;
	
	
	//================Alternative======================
	//fb_Warehouse_Modbus :ARRAY[0..3] OF FB_CommunicateModbusRTU; //0&1 : warehouse A , 2&3 : warehouse B
		//Declared in GVL due to Error handling request
	I		:UINT;
	SensorState	: ARRAY[0..99] OF BOOL;
	SensorStatesAll : un_RS485States_all;
	arr485sensor					: ARRAY [0..399] OF BOOL;
	fb_Warehouse_Modbus : ARRAY [0..3] OF FB_CommunicateModbusRTU;
	bMotorCoreUpdated	:	BOOL := TRUE;
	bReset				:	BOOL;
END_VAR

//M_CommunicateModbusRTU(bReset:=GVL.Reset,
//						bModBusRTUError=>bModbusRTUError,
//						udiModbusRTUErrorID=>udiModbusRTUErrorID);
						
//GVL.fbModbusRTUErrorTrans(
//	xDone:= , 
//	xBusy:= , 
//	xError:= bModbusRTUError, 
//	xAborted:= , 
//	iErrorID:= udiModbusRTUErrorID, 
//	Name:= 'Communicate ModBus RTU ');
	
	
	
//=================Alternative======================================
//Update FBs
bPassModBusMaster[0] := (*GVL_HMI.Setup.Mechanical.stModbusByPass.switchOff_1 OR*) GVL_Machine.stModbusByPassInternal.switchOff_1;
bPassModBusMaster[1] := (*GVL_HMI.Setup.Mechanical.stModbusByPass.switchOff_2 OR*) GVL_Machine.stModbusByPassInternal.switchOff_2;
bPassModBusMaster[2] := (*GVL_HMI.Setup.Mechanical.stModbusByPass.switchOff_3 OR*) GVL_Machine.stModbusByPassInternal.switchOff_3;
bPassModBusMaster[3] := (*GVL_HMI.Setup.Mechanical.stModbusByPass.switchOff_4 OR*) GVL_Machine.stModbusByPassInternal.switchOff_4;

//Update FBs
FOR I :=0 TO 3 BY 1 DO
	fb_Warehouse_Modbus[I](Execute:=bMotorCoreUpdated AND NOT bPassModBusMaster[I] , 
							   unitID :=UINT_TO_BYTE(I)+1 , 
							   Reset:=bReset,
							   MBdata_Read_ControllerN :=MBdata_Read_ControllerN[I],
							   ObjectName:=CONCAT('Communicate ModBus RTU : ',UINT_TO_STRING(I)),
							   arrSensor=>SensorStatesAll.arrSensorByController[I]);
	
	arr485sensor := SensorStatesAll.arrSensorAll;
	
END_FOR


//bPassModBusMaster[0] := GVL.stModbusByPass.switchOff_1;
//bPassModBusMaster[1] := GVL.stModbusByPass.switchOff_2;
//bPassModBusMaster[2] := GVL.stModbusByPass.switchOff_3;
//bPassModBusMaster[3] := GVL.stModbusByPass.switchOff_4;

END_PROGRAM

// ---- POUs/ModbusRTU/SerialComTask/FB_CommunicateModbusRTU.TcPOU
FUNCTION_BLOCK FB_CommunicateModbusRTU EXTENDS FB_ObjectBase_V2
VAR_INPUT
//    Execute    :BOOL;   // True : This prog will start.
//    Abort      :BOOL;   // True : This prog will be abort.
//    Reset      :BOOL;   // True : This prog will be reset.
//    ObjectName :STRING; // Set this fb name(About it's action)
	  
	  
	  unitID	  :BYTE;
	  MBdata_Read_ControllerN	: REFERENCE TO 	ARRAY[0..21] OF BYTE;
END_VAR

VAR_OUTPUT
//    Busy    :BOOL;        // True : This prog is running.
//    Done    :BOOL;        // True : Command has been executed.
//    Aborted :BOOL;        // True : This prog is aborted.
//    Error   :BOOL;        // True : This prog has an error.
//    ErrorID :UINT;       // Output ErrorID
//    Status  :T_MaxString; // Output this prog status by string(255bytes)
	arrSensor		: ARRAY[0..99] OF BOOL;
END_VAR

VAR
//    eState :E_MethodStatus_Basic;
//	uiExecutingStep : UDINT; // This var is used to been controll STATE_EXECUTING process.
//	uiResettingStep : UDINT;
//	uiAbortingStep : UDINT;
//	_Executed :BOOL; // Executing process completed.
//	_Error : BOOL; // FB has an error.
//	_ResetCompleted : BOOL; // FB resetting completed.
//	_AbortCompleted : BOOL; // FB aborting completed.
//	_Abort		: BOOL;
	strStatus	: STRING;
	uiResumeStep : UINT;
	arrSensorEmpty : ARRAY[0..99] OF BOOL;
	MB_EL6X22B_ControllerN	: ModbusRtuMasterV2_KL6x22B;
	fbComReset_ControllerN	: ComReset;	
	fbClearComBuffer		: ClearComBuffer;
	SensorState : un_RS485States;
	bComReset	:BOOL;
	bComResetBusy :BOOL;
	bComResetError :BOOL;
	bFB_ErrorOccur :BOOL;
END_VAR

A00_BasicUnits();
SUPER^.A10_StateControl();

ACTION A00_BasicUnits:
MB_EL6X22B_ControllerN();
fbComReset_ControllerN(
		Execute:= bComReset, 
		pComIn:= ADR(MB_EL6X22B_ControllerN.InData), 
		pComOut:= ADR(MB_EL6X22B_ControllerN.OutData), 
		SizeComIn:= SIZEOF(MB_EL6X22B_ControllerN.InData), 
		Done=> , 
		Busy=> bComResetBusy, 
		Error=> bComResetError, 
		ErrorID=> );
END_ACTION

METHOD GetModelState
VAR_OUTPUT
    xDone    :BOOL;
    xBusy    :BOOL;
    xError   :BOOL;
    xAborted :BOOL;
    iErrorID :UDINT;
	UniqueErrorCode : STRING;
END_VAR
xDone    := Done;
xBusy    := Busy;
xError   := Error;
xAborted := Abort;
iErrorID := ErrorID;
END_METHOD

METHOD GetName : STRING
GetName := ObjectName;
END_METHOD

METHOD PRIVATE M_AnalyzeData : BOOL
VAR_INPUT
	Data : ARRAY [0..21] OF BYTE;
END_VAR

VAR_OUTPUT
	arrSensor : ARRAY[0..9] OF BOOL;
END_VAR

arrSensor[0] :=Data[4].1;
arrSensor[1] :=Data[4].0;
arrSensor[2] :=Data[3].7;
arrSensor[3] :=Data[3].6;
arrSensor[4] :=Data[3].5;
arrSensor[5] :=Data[3].4;
arrSensor[6] :=Data[3].3;
arrSensor[7] :=Data[3].2;
arrSensor[8] :=Data[3].1;
arrSensor[9] :=Data[3].0;
END_METHOD

METHOD  M_STATE_ABORTED
VAR_INPUT
END_VAR
ERROR :=TRUE;
Busy    := FALSE;
Aborted := TRUE;
Status := strStatus;

IF NOT Execute THEN
	eSTATE:=STATE_RESETTING;
END_IF

IF Execute AND Reset THEN
	uiExecutingStep :=uiResumeStep;
	eSTATE:=STATE_EXECUTING;
END_IF
END_METHOD

METHOD  M_STATE_ABORTING
VAR_INPUT
END_VAR
CASE uiAbortingStep OF
	0 :
		uiAbortingStep:=9999;
	
	9999:	_AbortCompleted:=TRUE;
END_CASE

IF _AbortCompleted THEN	
	eSTATE :=STATE_ABORTED;
END_IF
END_METHOD

METHOD  M_STATE_DONE
VAR_INPUT
END_VAR
Busy 	:= FALSE;
Done	:=TRUE;

IF NOT Execute THEN
	eSTATE:=STATE_RESETTING;
END_IF
END_METHOD

METHOD  M_STATE_DORMANT
VAR_INPUT
END_VAR
Busy            := FALSE;
Done            := FALSE;
Aborted         := FALSE;
Error           := FALSE;
ErrorID         := 0;
Status          := '';
_ResetCompleted := FALSE;
_Error          := FALSE;
_Executed       := FALSE;
strStatus :='No Error';
uiExecutingStep :=uiResettingStep :=uiResumeStep :=0;
bComReset		:= FALSE;

arrSensor :=arrSensorEmpty;
// output all false if program stop working

IF Execute THEN
	eSTATE:=STATE_EXECUTING;
END_IF
END_METHOD

METHOD  M_STATE_ERROR
VAR_INPUT
END_VAR

VAR
	tempStr	:	STRING ;
END_VAR
ERROR   :=TRUE;
Busy	:=FALSE;
tempStr := CONCAT( 'Controllor ' , BYTE_TO_STRING(unitID));
Status := CONCAT(tempStr, strStatus);
ErrorID := unitID + 2600;// Start from 2600

IF NOT Execute OR Reset	THEN	
	eSTATE:=STATE_RESETTING;
END_IF
END_METHOD

METHOD  M_STATE_EXECUTING
VAR_INPUT
END_VAR

VAR
	arrSensorSingleModule : ARRAY [0..9] OF BOOL;	
	pMemoryAddr : ARRAY[0..7] OF BYTE;
END_VAR

VAR_INST
	Quantity : WORD;
	cbLength : UINT;
	
	iReadMBAddr :  WORD :=0;
END_VAR
Busy :=TRUE;
IF  MB_EL6X22B_ControllerN.Error AND NOT bFB_ErrorOccur  THEN
	bFB_ErrorOccur :=TRUE;
	_Error :=TRUE;
	strStatus :=' Modbus connection error';
END_IF

arrSensor:=SensorState.arrSensorByController;

IF iReadMBAddr <= 900 THEN
		Quantity :=10;	
	    cbLength :=20;
		MB_EL6X22B_ControllerN.ReadCoils();
ELSE
		Quantity :=1;
		cbLength :=2;
		MB_EL6X22B_ControllerN.ReadInputRegs();
END_IF

CASE uiExecutingStep OF
	
0: // Init
	MB_EL6X22B_ControllerN.Execute:=FALSE;
	iReadMBAddr:=0;
	uiExecutingStep:=100;
	
100:	
	MB_EL6X22B_ControllerN.UnitID:= unitID;
	MB_EL6X22B_ControllerN.Quantity:= Quantity; 
	MB_EL6X22B_ControllerN.MBAddr:= iReadMBAddr; 
	MB_EL6X22B_ControllerN.cbLength:= cbLength;
	MB_EL6X22B_ControllerN.pMemoryAddr:=ADR(pMemoryAddr) ; 
	MB_EL6X22B_ControllerN.Timeout:= T#1000MS; 
	MB_EL6X22B_ControllerN.Execute:=TRUE;	
	IF MB_EL6X22B_ControllerN.BUSY THEN
		uiExecutingStep:=200;
	END_IF	
	IF bFB_ErrorOccur THEN
		uiExecutingStep:=110;		
	END_IF
	
110:
	bFB_ErrorOccur :=FALSE; //Internal error flag 
	IF MB_EL6X22B_ControllerN.BUSY THEN
		uiExecutingStep:=200;
	END_IF
		
200:
	IF NOT MB_EL6X22B_ControllerN.BUSY THEN
		MB_EL6X22B_ControllerN.Execute:=FALSE;
		
		IF iReadMBAddr>=1000 THEN
			// Error checking step			
			IF MBdata_Read_ControllerN[1] = 4 AND MBdata_Read_ControllerN[3] + MBdata_Read_ControllerN[4] > 0 THEN
				_Error := TRUE;
				strStatus :=' Controller report error';
			END_IF
			
			iReadMBAddr :=0;
			
		ELSE
			// Signal step
			M_AnalyzeData(Data :=MBdata_Read_ControllerN,arrSensor=>arrSensorSingleModule);
			SensorState.arrSensorBySingleModule[iReadMBAddr/100] :=arrSensorSingleModule;		
			iReadMBAddr :=iReadMBAddr +100;
		END_IF
		
		uiExecutingStep:=100;		
		
	 END_IF

END_CASE
	
IF NOT Execute THEN
	eState:=STATE_RESETTING;
END_IF
IF _Error THEN
	eState:=STATE_ERROR;
END_IF
IF _Abort THEN
	eSTATE:=STATE_ABORTING;
END_IF
IF _Executed THEN
	eSTATE:=STATE_Done;
END_IF
END_METHOD

METHOD  M_STATE_RESETTING
VAR_INPUT
END_VAR
Error :=FALSE;
Done :=FALSE;
Busy := FALSE;


CASE uiResettingStep OF
	
	0:
		MB_EL6X22B_ControllerN.Execute:=FALSE;
//		fbClearComBuffer(Buffer:=MB_EL6X22B_ControllerN.InData);
//		fbClearComBuffer(Buffer:=MB_EL6X22B_ControllerN.OutData);
		uiResettingStep:=100;
	100:	
		bComReset := TRUE;
		IF fbComReset_ControllerN.Busy THEN
			uiResettingStep:=200;
		END_IF
	200:
		IF fbComReset_ControllerN.Done THEN
			uiResettingStep:=9999;
		END_IF

	9999:
		_Error:=FALSE;
		_ResetCompleted:=TRUE;
END_CASE
IF _ResetCompleted THEN
	eSTATE:=STATE_DORMANT;
END_IF
END_METHOD

END_FUNCTION_BLOCK

// ---- Library/10_Machine/00_BaseFBs/01_FB_ObjectBase/FB_ObjectBase_V2.TcPOU
FUNCTION_BLOCK FB_ObjectBase_V2 IMPLEMENTS IBasicElement
VAR_INPUT
    Execute    	: BOOL;   // True : This prog will start.
    Abort      	: BOOL;   // True : This prog will be abort.
    Reset      	: BOOL;   // True : This prog will be reset.
	Pause	   	: BOOL;
    ObjectName 	: STRING; // Set this fb name(About it's action)
END_VAR

VAR_OUTPUT
    Busy    	: BOOL;        // True : This prog is running.
    Done    	: BOOL;        // True : Command has been executed.
    Aborted 	: BOOL;        // True : This prog is aborted.
    Error   	: BOOL;        // True : This prog has an error.
	Paused		: BOOL;
    ErrorID 	: UINT;       // Output ErrorID
    Status  	: STRING; // Output this prog status by string(255bytes)
	UniqueErrorCode :STRING;	
END_VAR

VAR
    eState :E_MethodStatus_Basic;
	uiExecutingStep : UDINT; // This var is used to been controll STATE_EXECUTING process.
	uiResettingStep : UDINT;
	uiAbortingStep  : UDINT;
	
	// Pause Step
	uiHoldingStep	: UDINT;
	uiHeldStep		: UDINT;
	uiUnholdStep	: UDINT;
	
	_Executed 	: BOOL; // Executing process completed.
	_Error 		: BOOL; // FB has an error.
	_Abort		: BOOL;
	
	_ResetCompleted 	: BOOL; // FB resetting completed.
	_AbortCompleted 	: BOOL; // FB aborting completed.
	_HoldingCompleted	: BOOL;
	_HeldCompleted		: BOOL;
	_UnholdCompleted	: BOOL;		
END_VAR

A00_BasicUnits();
A10_StateControl();

ACTION A00_BasicUnits:

END_ACTION

ACTION A10_StateControl:
CASE eState OF
	STATE_DORMANT:
		M_STATE_DORMANT();
	STATE_EXECUTING:
		M_STATE_EXECUTING();
	STATE_ABORTING:
		M_STATE_ABORTING();
	STATE_ABORTED:
		M_STATE_ABORTED();
	STATE_DONE:
		M_STATE_DONE();
	STATE_ERROR:
		M_STATE_ERROR();
	STATE_RESETTING:
		M_STATE_RESETTING();
	STATE_Holding:
		M_STATE_HOLDING();
	STATE_Held:
		M_STATE_HELD();
	STATE_UnHold:
		M_STATE_UNHOLD();
END_CASE
END_ACTION

METHOD GetModelState
VAR_OUTPUT
    xDone    :BOOL;
    xBusy    :BOOL;
    xError   :BOOL;
    xAborted :BOOL;
    iErrorID :UDINT;	
	UniqueErrorCode : STRING;
END_VAR
xDone    := Done;
xBusy    := Busy;
xError   := Error;
xAborted := Abort;
iErrorID := ErrorID;
UniqueErrorCode := THIS^.UniqueErrorCode;
END_METHOD

METHOD GetName : STRING
GetName := ObjectName;
END_METHOD

METHOD M_FormatManagedStatus : STRING
VAR_INPUT
    AlarmId : DINT;
    InnerMessage : STRING;
END_VAR
VAR
    sPrefix : STRING;
END_VAR
sPrefix := CONCAT('[', DINT_TO_STRING(AlarmId));
sPrefix := CONCAT(sPrefix, '-');
sPrefix := CONCAT(sPrefix, UDINT_TO_STRING(uiExecutingStep));
sPrefix := CONCAT(sPrefix, '] ');
M_FormatManagedStatus := CONCAT(sPrefix, InnerMessage);
END_METHOD

METHOD M_RefLinks
VAR_INPUT
END_VAR
END_METHOD

METHOD  M_STATE_ABORTED
VAR_INPUT
END_VAR
;

(*

Busy  := FALSE;
Error := TRUE;
Aborted := TRUE;
uiAbortingStep 	:= 0;
_AbortCompleted := FALSE;

// 狀態機切換
IF NOT Execute THEN
	eState := STATE_RESETTING;
ELSIF Execute AND reset THEN
	Error	:= false;
	Aborted	:= false;
	eState 	:= STATE_EXECUTING;
END_IF

*)
END_METHOD

METHOD  M_STATE_ABORTING
VAR_INPUT
END_VAR
;
(*


CASE uiAbortingStep OF
	0 :
		_Abort := false;
		uiAbortingStep:=9999;

	9999:	
		_AbortCompleted:=TRUE;
END_CASE

IF _AbortCompleted THEN	
	eSTATE :=STATE_ABORTED;
END_IF

*)
END_METHOD

METHOD  M_STATE_DONE
VAR_INPUT
END_VAR
;

(*

Busy := FALSE;
Done := TRUE;
IF NOT Execute THEN
    eState := STATE_RESETTING;
END_IF

*)
END_METHOD

METHOD  M_STATE_DORMANT
VAR_INPUT
END_VAR
;

(*
Busy 			:= FALSE;
Done 			:= FALSE;
Aborted 		:= FALSE;
Error			:= FALSE;
Paused			:= FALSE;
ErrorID			:= 0;
Status			:= '';
UniqueErrorCode := '';

_Executed 			:= FALSE;
_Error				:= FALSE;
_Abort				:= FALSE;
_ResetCompleted 	:= FALSE;
_AbortCompleted 	:= FALSE;
_HoldingCompleted 	:= FALSE;
_HeldCompleted	 	:= FALSE;
_UnholdCompleted 	:= FALSE;

uiExecutingStep 		:= 0;
uiResettingStep 		:= 0;
uiAbortingStep 			:= 0;
uiHoldingStep			:= 0;
uiHeldStep				:= 0;
uiUnholdStep			:= 0;

IF Execute THEN
    eState := STATE_EXECUTING;
END_IF
*)
END_METHOD

METHOD  M_STATE_ERROR
VAR_INPUT
END_VAR
;

(*
ERROR   := TRUE;
Busy	:= FALSE;
_Error	:= false;

IF NOT Execute THEN	
	Error	:= false;
	eSTATE	:=STATE_RESETTING;
END_IF

*)
END_METHOD

METHOD  M_STATE_EXECUTING
VAR_INPUT
END_VAR
;

(*
busy := true;

// 暫停
IF Pause THEN 
	_HoldingCompleted 	:= FALSE;
	_HeldCompleted	 	:= FALSE;
	_UnholdCompleted 	:= FALSE;
	uiHoldingStep		:= 0;
	uiHeldStep			:= 0;
	uiUnholdStep		:= 0;
	eState    			:= STATE_Holding;
END_IF

// 動作主流程 狀態機
case uiExecutingStep of

end_case

// 狀態機切換
IF NOT Execute THEN
	eState := STATE_RESETTING;
ELSIF _Error THEN
	eState := STATE_ERROR;
ELSIF _Abort THEN
	eState := STATE_ABORTING;
ELSIF _Executed THEN
	eState := STATE_DONE;
END_IF
	
*)
END_METHOD

METHOD M_STATE_HELD
VAR_INPUT
END_VAR
;
(*

Busy 	:= FALSE;
Paused 	:= TRUE;

CASE uiHeldStep OF
	0:
		uiHeldStep := 9999;

	9999:
		_HeldCompleted := TRUE;	

END_CASE

IF _HeldCompleted AND NOT Pause THEN
	eState := STATE_UnHold;
END_IF

*)
END_METHOD

METHOD M_STATE_HOLDING
VAR_INPUT
END_VAR
;

(*

CASE uiHoldingStep OF 
	0:	    // 需關閉 Timer 等等須暫停的變數
		uiHoldingStep := 9999;
		
	9999:	// holding 完成
		_HoldingCompleted := TRUE;
END_CASE

IF _HoldingCompleted THEN
	eState := STATE_Held;
END_IF

*)
END_METHOD

METHOD  M_STATE_RESETTING
VAR_INPUT
END_VAR
;

(*

CASE uiResettingStep OF
	
	0:
		uiResettingStep := 9999;
	9999:
		_ResetCompleted:=TRUE;
END_CASE

IF _ResetCompleted THEN
	eSTATE:=STATE_DORMANT;
END_IF

*)
END_METHOD

METHOD M_STATE_UNHOLD
VAR_INPUT
END_VAR
;
(*

CASE uiUnholdStep OF 
	0:		
		uiUnholdStep := 9999;
		
	9999:
		_UnholdCompleted := TRUE;
		
END_CASE

IF _UnholdCompleted THEN
	Paused := FALSE;
	eState := STATE_EXECUTING;
END_IF

*)
END_METHOD

END_FUNCTION_BLOCK

// ---- POUs/RS485_JidianVersion/MAIN2_RS485.TcPOU
PROGRAM MAIN2_RS485
VAR
	RS485_V2:ARRAY[1..4] OF FB_WarehouseSensorCtrl;
	
	i	: INT := 1;
	j	: INT;
	k	: INT;
	arr485sensor					: ARRAY [1..400] OF BOOL;

END_VAR

RS485_V2[1](bEnable:=TRUE);
RS485_V2[2](bEnable:=TRUE,UnitID := 2);
RS485_V2[3](bEnable:=TRUE,UnitID := 3);
RS485_V2[4](bEnable:=TRUE,UnitID := 4);

RS485_V2[1].ErrorId;
RS485_V2[2].ErrorId;
RS485_V2[3].ErrorId;
RS485_V2[4].ErrorId;

RS485_V2[1].RS485_ErrorCount;
RS485_V2[2].RS485_ErrorCount;
RS485_V2[3].RS485_ErrorCount;
RS485_V2[4].RS485_ErrorCount;

FOR i := 1 TO 400 DO
	k := i MOD 100;
	IF k = 0 THEN
		j := i/100;
		k := 100;
	ELSE
		j := (i/100) + 1;
	END_IF
	arr485sensor[i]:= RS485_V2[j].stRS485Controller.stSliderStatusALL.bPos[k];
END_FOR

END_PROGRAM

// ---- POUs/RS485_JidianVersion/FB_WarehouseSensorCtrl.TcPOU
FUNCTION_BLOCK FB_WarehouseSensorCtrl
VAR_INPUT
	bEnable: BOOL;
//	UnitID: INT:= 1; //AFU改
	UnitID: BYTE:= 1;  //AFU改
	nQuantity: INT:= 16;
	nMBAddr: INT;
END_VAR
VAR_OUTPUT
	bBusy: BOOL;
	bError: BOOL;
	ErrorId: MODBUS_ERRORS;
	ErrorMsg	:T_MaxString;
	stRS485Controller: ST_RS485Controller;
END_VAR
VAR
	stSliderStatusALL: ST_RS485_SliderStatusALL;
	stLayerStatus: ST_RS485_LayerStatus;
	stHeartbeat: ST_RS485_Heartbeat;
	ModbusRtuMasterV2_KL6x22B: ModbusRtuMasterV2_KL6x22B;
	//ModbusBIT: ModbusBIT;
	Data: ARRAY[0..9] OF WORD;
	Switch: INT;
	bEnableTest: BOOL;
	Count_Error: CTU;
	RS485_ErrorCount: WORD;
	bCheckHeartBitOnline	: BOOL;
	TON_checkHeart	: TON;
END_VAR
VAR CONSTANT
	nMBAddrMax: INT := 10;
END_VAR

TON_checkHeart(PT:=T#10S);
IF nMBAddr <= 0 THEN
	nMBAddr:= 0;
ELSIF nMBAddr >= 9 THEN
	nMBAddr:= 9;
END_IF
(*
CC(
	CU:= , 
	RESET:= , 
	PV:= , 
	Q=> , 
	CV=> );

*)


Count_Error(
	CU:= bError, 
	RESET:= , 
	PV:= 1000, 
	Q=> , 
	CV=> );
	
RS485_ErrorCount := Count_Error.CV;
	
	
	
IF bEnableTest THEN
	ModbusRtuMasterV2_KL6x22B.ReadCoils(
			UnitID:= UnitID, 
			Quantity:= nQuantity, 
			MBAddr:= nMBAddr * 100 , 
			cbLength:= nQuantity * 2 , 
			pMemoryAddr:= ADR(Data[nMBAddr]) , 
			AuxQuantity:= , 
			AuxMBAddr:= , 
			AuxcbLength:= , 
			pAuxMemoryAddr:= , 
			Execute:= , 
			Timeout:= T#1S, 
			BUSY=> bBusy, 
			Error=> , 
			ErrorId=> ErrorId, 
			cbRead=> );
END_IF



CASE Switch OF
	0:
		IF NOT bEnableTest THEN
			ModbusRtuMasterV2_KL6x22B.ReadCoils(
				UnitID:= UnitID, 
				Quantity:= nQuantity, 
				MBAddr:= nMBAddr * 100 , 
				cbLength:= nQuantity * 2 , 
				pMemoryAddr:= ADR(Data[nMBAddr]) , 
				AuxQuantity:= , 
				AuxMBAddr:= , 
				AuxcbLength:= , 
				pAuxMemoryAddr:= , 
				Execute:= FALSE, 
				Timeout:= T#1S, 
				BUSY=> bBusy, 
				Error=>, 
				ErrorId=> ErrorId, 
				cbRead=> );
			END_IF
		IF bEnable THEN
			Switch:= 100;
		END_IF
	100:
		ModbusRtuMasterV2_KL6x22B.ReadCoils(
			UnitID:= UnitID, 
			Quantity:= nQuantity, 
			MBAddr:= nMBAddr * 100 , 
			cbLength:= nQuantity * 2 , 
			pMemoryAddr:= ADR(Data[nMBAddr]) , 
			AuxQuantity:= , 
			AuxMBAddr:= , 
			AuxcbLength:= , 
			pAuxMemoryAddr:= , 
			Execute:= TRUE, 
			Timeout:= T#1S, 
			BUSY=> bBusy, 
			Error=> , 
			ErrorId=> ErrorId, 
			cbRead=> );
		IF ModbusRtuMasterV2_KL6x22B.BUSY THEN
			ModbusRtuMasterV2_KL6x22B.ReadCoils(Execute:= FALSE);
			Switch:=Switch+10;
		END_IF	
	110:
		ModbusRtuMasterV2_KL6x22B.ReadCoils(Execute:= FALSE ,Timeout:=T#1S ,BUSY=>bBusy ,Error=> ,ErrorId=>ErrorId ,);	
		IF NOT ModbusRtuMasterV2_KL6x22B.BUSY AND NOT ModbusRtuMasterV2_KL6x22B.Error THEN
			Switch:= 200;
		ELSIF ModbusRtuMasterV2_KL6x22B.Error THEN
			Switch:= 0;
		END_IF
	200:
		IF nMBAddr < (nMBAddrMax - 1) THEN
			nMBAddr:= nMBAddr + 1;
		ELSE
			nMBAddr:= 0;
		END_IF
		Switch:= 500;
	500:
		IF bEnable THEN
			Switch:= 100;
		ELSE
			Switch:= 0;
		END_IF
END_CASE	
		

	stHeartbeat.nHeartbeat1:= Data[0].10;
	stHeartbeat.nHeartbeat2:= Data[1].11;
	stHeartbeat.nHeartbeat3:= Data[2].10 AND Data[2].11;
	stHeartbeat.nHeartbeat4:= Data[3].12;
	stHeartbeat.nHeartbeat5:= Data[4].10 AND Data[4].12;
	stHeartbeat.nHeartbeat6:= Data[5].11 AND Data[5].12;
	stHeartbeat.nHeartbeat7:= Data[6].10 AND Data[6].11 AND Data[6].12;
	stHeartbeat.nHeartbeat8:= Data[7].13;
	stHeartbeat.nHeartbeat9:= Data[8].10 AND Data[8].13;
	stHeartbeat.nHeartbeat10:= Data[9].11 AND Data[9].13;
	
	bCheckHeartBitOnline := stHeartbeat.nHeartbeat1 AND
							stHeartbeat.nHeartbeat2 AND
							stHeartbeat.nHeartbeat3 AND
							stHeartbeat.nHeartbeat4 AND
							stHeartbeat.nHeartbeat5 AND
							stHeartbeat.nHeartbeat6 AND
							stHeartbeat.nHeartbeat7 AND
							stHeartbeat.nHeartbeat8 AND
							stHeartbeat.nHeartbeat9 AND 
							stHeartbeat.nHeartbeat10;
	
	TON_checkHeart.IN := NOT bCheckHeartBitOnline;
	IF TON_checkHeart.Q THEN
//		bError := TRUE;
		ErrorMsg := 'ModBus RTU heartBit not Online ,please ';
	ELSE
		ErrorMsg := '';
	END_IF
	
	bError := TON_checkHeart.Q OR ModbusRtuMasterV2_KL6x22B.Error;
							
	(*
	stLayerStatus.PCB1:=NOT ModbusBIT.b1001;
	stLayerStatus.PCB2:=NOT ModbusBIT.b1002;
	stLayerStatus.PCB3:=NOT ModbusBIT.b1003;
	stLayerStatus.PCB4:=NOT ModbusBIT.b1004;
	stLayerStatus.PCB5:=NOT ModbusBIT.b1005;
	stLayerStatus.PCB6:=NOT ModbusBIT.b1006;
	stLayerStatus.PCB7:=NOT ModbusBIT.b1007;
	stLayerStatus.PCB8:=NOT ModbusBIT.b1008;
	stLayerStatus.PCB9:=NOT ModbusBIT.b1009;
	stLayerStatus.PCB10:=NOT ModbusBIT.b1010;
	*)
	
	 stSliderStatusALL.bPos[10]:=Data[0].0;
	 stSliderStatusALL.bPos[9]:=Data[0].1;
	 stSliderStatusALL.bPos[8]:=Data[0].2;
	 stSliderStatusALL.bPos[7]:=Data[0].3;
	 stSliderStatusALL.bPos[6]:=Data[0].4;
	 stSliderStatusALL.bPos[5]:=Data[0].5;
	 stSliderStatusALL.bPos[4]:=Data[0].6;
	 stSliderStatusALL.bPos[3]:=Data[0].7;
	 stSliderStatusALL.bPos[2]:=Data[0].8;
	 stSliderStatusALL.bPos[1]:=Data[0].9;
	 
	 stSliderStatusALL.bPos[20]:=Data[1].0;
	 stSliderStatusALL.bPos[19]:=Data[1].1;
	 stSliderStatusALL.bPos[18]:=Data[1].2;
	 stSliderStatusALL.bPos[17]:=Data[1].3;
	 stSliderStatusALL.bPos[16]:=Data[1].4;
	 stSliderStatusALL.bPos[15]:=Data[1].5;
	 stSliderStatusALL.bPos[14]:=Data[1].6;
	 stSliderStatusALL.bPos[13]:=Data[1].7;
	 stSliderStatusALL.bPos[12]:=Data[1].8;
	 stSliderStatusALL.bPos[11]:=Data[1].9;
	 
	 stSliderStatusALL.bPos[30]:=Data[2].0;
	 stSliderStatusALL.bPos[29]:=Data[2].1;
	 stSliderStatusALL.bPos[28]:=Data[2].2;
	 stSliderStatusALL.bPos[27]:=Data[2].3;
	 stSliderStatusALL.bPos[26]:=Data[2].4;
	 stSliderStatusALL.bPos[25]:=Data[2].5;
	 stSliderStatusALL.bPos[24]:=Data[2].6;
	 stSliderStatusALL.bPos[23]:=Data[2].7;
	 stSliderStatusALL.bPos[22]:=Data[2].8;
	 stSliderStatusALL.bPos[21]:=Data[2].9;
	 
	 stSliderStatusALL.bPos[40]:=Data[3].0;
	 stSliderStatusALL.bPos[39]:=Data[3].1;
	 stSliderStatusALL.bPos[38]:=Data[3].2;
	 stSliderStatusALL.bPos[37]:=Data[3].3;
	 stSliderStatusALL.bPos[36]:=Data[3].4;
	 stSliderStatusALL.bPos[35]:=Data[3].5;
	 stSliderStatusALL.bPos[34]:=Data[3].6;
	 stSliderStatusALL.bPos[33]:=Data[3].7;
	 stSliderStatusALL.bPos[32]:=Data[3].8;
	 stSliderStatusALL.bPos[31]:=Data[3].9;
	 
	 stSliderStatusALL.bPos[50]:=Data[4].0;
	 stSliderStatusALL.bPos[49]:=Data[4].1;
	 stSliderStatusALL.bPos[48]:=Data[4].2;
	 stSliderStatusALL.bPos[47]:=Data[4].3;
	 stSliderStatusALL.bPos[46]:=Data[4].4;
	 stSliderStatusALL.bPos[45]:=Data[4].5;
	 stSliderStatusALL.bPos[44]:=Data[4].6;
	 stSliderStatusALL.bPos[43]:=Data[4].7;
	 stSliderStatusALL.bPos[42]:=Data[4].8;
	 stSliderStatusALL.bPos[41]:=Data[4].9;
	 
	 stSliderStatusALL.bPos[60]:=Data[5].0;
	 stSliderStatusALL.bPos[59]:=Data[5].1;
	 stSliderStatusALL.bPos[58]:=Data[5].2;
	 stSliderStatusALL.bPos[57]:=Data[5].3;
	 stSliderStatusALL.bPos[56]:=Data[5].4;
	 stSliderStatusALL.bPos[55]:=Data[5].5;
	 stSliderStatusALL.bPos[54]:=Data[5].6;
	 stSliderStatusALL.bPos[53]:=Data[5].7;
	 stSliderStatusALL.bPos[52]:=Data[5].8;
	 stSliderStatusALL.bPos[51]:=Data[5].9;
	 
	 stSliderStatusALL.bPos[70]:=Data[6].0;
	 stSliderStatusALL.bPos[69]:=Data[6].1;
	 stSliderStatusALL.bPos[68]:=Data[6].2;
	 stSliderStatusALL.bPos[67]:=Data[6].3;
	 stSliderStatusALL.bPos[66]:=Data[6].4;
	 stSliderStatusALL.bPos[65]:=Data[6].5;
	 stSliderStatusALL.bPos[64]:=Data[6].6;
	 stSliderStatusALL.bPos[63]:=Data[6].7;
	 stSliderStatusALL.bPos[62]:=Data[6].8;
	 stSliderStatusALL.bPos[61]:=Data[6].9;
	 
	 stSliderStatusALL.bPos[80]:=Data[7].0;
	 stSliderStatusALL.bPos[79]:=Data[7].1;
	 stSliderStatusALL.bPos[78]:=Data[7].2;
	 stSliderStatusALL.bPos[77]:=Data[7].3;
	 stSliderStatusALL.bPos[76]:=Data[7].4;
	 stSliderStatusALL.bPos[75]:=Data[7].5;
	 stSliderStatusALL.bPos[74]:=Data[7].6;
	 stSliderStatusALL.bPos[73]:=Data[7].7;
	 stSliderStatusALL.bPos[72]:=Data[7].8;
	 stSliderStatusALL.bPos[71]:=Data[7].9;
	 
	 stSliderStatusALL.bPos[90]:=Data[8].0;
	 stSliderStatusALL.bPos[89]:=Data[8].1;
	 stSliderStatusALL.bPos[88]:=Data[8].2;
	 stSliderStatusALL.bPos[87]:=Data[8].3;
	 stSliderStatusALL.bPos[86]:=Data[8].4;
	 stSliderStatusALL.bPos[85]:=Data[8].5;
	 stSliderStatusALL.bPos[84]:=Data[8].6;
	 stSliderStatusALL.bPos[83]:=Data[8].7;
	 stSliderStatusALL.bPos[82]:=Data[8].8;
	 stSliderStatusALL.bPos[81]:=Data[8].9;
	 
	 stSliderStatusALL.bPos[100]:=Data[9].0;
	 stSliderStatusALL.bPos[99]:=Data[9].1;
	 stSliderStatusALL.bPos[98]:=Data[9].2;
	 stSliderStatusALL.bPos[97]:=Data[9].3;
	 stSliderStatusALL.bPos[96]:=Data[9].4;
	 stSliderStatusALL.bPos[95]:=Data[9].5;
	 stSliderStatusALL.bPos[94]:=Data[9].6;
	 stSliderStatusALL.bPos[93]:=Data[9].7;
	 stSliderStatusALL.bPos[92]:=Data[9].8;
	 stSliderStatusALL.bPos[91]:=Data[9].9;	
	 
	stRS485Controller.stSliderStatusALL:=stSliderStatusALL;
	stRS485Controller.stLayerStatus:=stLayerStatus;
	stRS485Controller.stHeartbeat:=stHeartbeat;

END_FUNCTION_BLOCK

// ---- Library/10_Machine/12_MachineControl/FB_MachineControl.TcPOU
FUNCTION_BLOCK FB_MachineControl EXTENDS FB_ModeBase_V2 IMPLEMENTS I_UnitState
VAR_INPUT
    INPUT            : REFERENCE TO ST_InputTable;
    OUTPUT           : REFERENCE TO ST_OutputTable;
    EnableSimulation : BOOL       := FALSE	;
    DataDirect       : E_DataFrom := E_DataFrom.Remote;
END_VAR
VAR_OUTPUT
    Error               : BOOL;
    ErrorID             : DINT;
    ErrMsg              : T_MaxString;
    CylinderStatus      : ST_CylinderStatus;
    MotorStatus         : ST_MotorStatus;
    StorageRobot_EStop  : BOOL;
    ShippingRobot_EStop : BOOL;
    MachineHomed        : BOOL;
    // Machine OpPannel 
    Machine_Estop : BOOL;
    Machine_Start : BOOL;
    Machine_Stop  : BOOL;
    Machine_Reset : BOOL;
	// 提供給手臂Service 下達清理錯誤命令
	RobotService_ResetCmd	: BOOL;		// 兩個旗標都由Service資料夾內的Method 控制
	RobotService_StartCmd	: BOOL;
	ShippingRobotService_ResetCmd	: BOOL;	// 提供給出貨區手臂，清除手臂錯誤
	ShippingRobotService_StartCmd	: BOOL;
END_VAR
VAR
    // C# HMI handshake
    fbHmiHandShakeController : FB_HmiHandShake;

    // internal Output
    InternalOutput : ST_OutputTable;

    // Componets setup parameter
    CurrentData : ST_SetupPara;

    // Current Manual Command
    AllocateManualCommand   : ST_Manual_Allocated;
    StorageManualCommand    : ST_Manual_Storage;
    ShippingManualCommand   : ST_Manual_Shipping;
    AllocateHalfAutoCommand : REFERENCE TO ST_HalfAuto_Allocated;
    // Area controller
    fbAllocateArea : FB_AllocateAreaWithRoundbelt;
    fbStorageArea  : FB_StorageArea;
    fbShippingArea : FB_ShippingArea;

    // Service controller
    TableMove : FB_TableMove;
	fbMachineHoming : FB_MachineHoming;
    // Componets
    Cylinder           : UNI_CylinderList;
    Motor              : UNI_MotorList;
    FanucRobot         : UNI_FanucRobotList;
    // 同尺寸軌道仲裁 request (Phase 2 集中式 motor control,各 sub-FB 寫請求,由 A20_ConveyorArbitration 仲裁)
    SameSizeCVRequest  : ST_SameSizeCVRequest;
    // 一次性 latch:首次 ShippingPlateScan 觸發時 Press1 / Press3 伸出擋盒,之後 FB_ShippingPlateScan 不再重伸 (避免每次都動造成問題)。FALSE 預設,PLC boot 後第一次 ShippingScan 自動 latch 為 TRUE。
    bSameSizeCV_Press1_AlreadyExtended : BOOL;
    bSameSizeCV_Press3_AlreadyExtended : BOOL;
    CylinderManualCtrl : ARRAY[1..udiMax_CylinderNum] OF FB_CylinderManualCtrl;
	MotorManualCtrl    : ARRAY[1..26] OF 	FB_MotorManualCtrl;
    // Wheelhouse Sensor
    WheelhouseSensor : UNI_HMI_WheelHouseInput;

    bCheckMotorWork   : BOOL;
    Service_Handshake : ST_HMI_Handshake; // To read legacy HMI data
    StorageService    : ST_StorageService;
    AllocateService   : ST_AllocateService;
    ShippingService   : ST_ShippingService;
	
    Allocate_EStop			: BOOL;
    Storage_EStop  			: BOOL;
	Allocate_EStopEdgeDetect : FB_EdgeDetect;
    Storage_EstopEdgeDetect  : FB_EdgeDetect;
	
	bStorage_AirPressure 	: BOOL;
	// ErrorHandler
	fbErrorHandler 		:FB_ErrorHandler_V2;
	ErrorTableInitDone 	: BOOL;
	E_StopEdgeDetect	: FB_EdgeDetect;
	StartEdgeDetect 	: FB_EdgeDetect;
	ResetEdgeDetect 	: FB_EdgeDetect;
	StopEdgeDetect 		: FB_EdgeDetect;
	bSafetyDoorOpen 	: BOOL;
	fbBlink_05 			: BLINK;
	bStopMem 			: BOOL;
    fb_AllocateSignalTower : FB_SignalTower;
    fb_StorageSignalTower  : FB_SignalTower;
	_RedLamp 			: BOOL;
	_YellowLamp			: BOOL;
	_GreenLamp 			: BOOL;
	_Buzz 				: BOOL;
	bTest2 				: BOOL;
	SafeDoorsOpen 		: ARRAY[0..20] OF BOOL;
	SafeDoorResetError	: BOOL;
	bStorageRobotError	: BOOL;
	bShippingRobotError	: BOOL;
	i 					: INT;
	BuzzCtrlUseBuzz		: BOOL;
	
	//Btn ctrl
	tofResetDelay	:TOF;
	tofStopDelay	:TOF;
	tofStartDelay	:TOF;
	
	tonDelayErrorHandle : TON;
	
	/// HMI storage camera blow ctrl    edit by min 20251031
	fbHmiCameraBlow		: FB_EdgeDetect;
	
	//Test bool signal with hans laser 
	bAsideComplete	: BOOL;
	bBsideComplete	: BOOL;
	
	ResetDetect		: BOOL;
	
	// 提供給手臂Service 下達清理錯誤命令
	TON_RobotReleaseResetCmd	: TON;
	TON_RobotReleaseStartCmd	: TON;
	TON_Shipping_RobotRelease_ResetCmd	: TON;
	TON_Shipping_RobotRelease_StartCmd	: TON;
	
	fbBuzzCtrl : FB_BuzzCtrl;
	fbMachineModeSwitch : FB_MachineModeSwitch;
    // 數位孿生 IO 模擬 FB
    fbSimulatedIO : FB_SimulatedIO;
	
END_VAR

// Implement PackML State Machine
SUPER^();
tonDelayErrorHandle(IN:=TRUE, PT:=T#5S); // Delay 5s after PLC run then check error
A00_BaseUnits();
A01_Cylinder();
A02_Motor();
A20_ConveyorArbitration();
A03_FanucRobot();
A04_OpPannel();
A05_Light();
IF tonDelayErrorHandle.Q THEN
	A10_ErrorHandler();
END_IF

IF NOT EnableSimulation THEN
    OUTPUT := InternalOutput;
ELSE
    OUTPUT := InternalOutput; // 模擬模式仍輸出（無實體硬體，安全無虞）；FB_SimulatedIO 才能讀到 Valve 狀態
    fbSimulatedIO(); // 注入安全輸入 + 汽缸感測器回饋
END_IF

//WheelhouseSensor.arWheelHouseInput := ComModbusRTU.arr485sensor;
WheelhouseSensor.arWheelHouseInput := MAIN2_RS485.arr485sensor;

IF DataDirect = E_DataFrom.Local THEN
    CurrentData := GVL_Machine.LocalData;
ELSIF DataDirect = E_DataFrom.Remote THEN
    CurrentData := GVL_Machine.RemoteData;
    AllocateManualCommand := GVL_HMI.Allocated.Manual;
    StorageManualCommand := GVL_HMI.Storage.Manual;
    ShippingManualCOmmand := GVL_HMI.Shipping.Manual;
    AllocateHalfAutoCommand REF= GVL_HMI.Allocated.HalfAuto;
END_IF
gvl_ads.MachineState := FUN_MachineState(
	Error:= xError, 
	Estop:= FALSE, 
	Stop:= Machine_Stop, 
	Reset:= Machine_Reset OR tofResetDelay.Q , 
	Start:= Machine_Start,
	eMachineState :=  gvl_ads.MachineState,
	HomeBusy:= fbMachineHoming.xBusy, 
	Homed:= MachineHomed, 
	MachineMode:= eModeCurrent);

ACTION A00_BaseUnits:
fbStorageArea(eModeCommand :=,
              eStateCommand :=,
			  FanucRobot := FanucRobot.List.StorageRobot,
              PackTag := GVL_Machine.PackTags[UnitNo.Storage],
			  Service := StorageService,
			  WheelhouseSensor :=WheelhouseSensor,
			  Motor := Motor,
			  Input := INPUT,
			  Output := InternalOutput,
			  Reset := Machine_Reset,
			  Stop := Machine_Stop,
			  bStopMem:=bStopMem,
			  Cylinder:= Cylinder,
			  CurrentData :=CurrentData,
              eModeCurrent => GVL_Machine.PackTags[UnitNo.Storage].Status.UnitModeCurrent,
              eStateCurrent => GVL_Machine.PackTags[UnitNo.Storage].Status.StateCurrent);

fbAllocateArea(eModeCommand :=,
               eStateCommand :=,
			   INPUT :=INPUT,
			   OUTPUT :=InternalOutput,
			   Cylinder := Cylinder,
			   Motor := Motor,
			   SameSizeCVRequest := SameSizeCVRequest,
			   Reset := Machine_Reset,
			   Stop := Machine_Stop,
			   bStopMem:=bStopMem,
			   CurrentData := CurrentData,
               PackTag := GVL_Machine.PackTags[UnitNo.Allocate],
			   service := AllocateService,
               eModeCurrent => GVL_Machine.PackTags[UnitNo.Allocate].Status.UnitModeCurrent,
               eStateCurrent => GVL_Machine.PackTags[UnitNo.Allocate].Status.StateCurrent);

fbShippingArea(eModeCommand :=,
               eStateCommand :=,
			   FanucRobot:= FanucRobot.List.ShippingRobot,
			   INPUT :=INPUT,
			   OUTPUT := InternalOutput,
			   Motor := Motor,
			   Cylinder := Cylinder,
			   SameSizeCVRequest := SameSizeCVRequest,
			   SameSizeCV_Press1_AlreadyExtended := bSameSizeCV_Press1_AlreadyExtended,
			   SameSizeCV_Press3_AlreadyExtended := bSameSizeCV_Press3_AlreadyExtended,
			   Reset := Machine_Reset,
			   Stop := Machine_Stop,
			   bStopMem:=bStopMem,
               PackTag := GVL_Machine.PackTags[UnitNo.Shipping],
			   Service := ShippingService,
               eModeCurrent => GVL_Machine.PackTags[UnitNo.Shipping].Status.UnitModeCurrent,
               eStateCurrent => GVL_Machine.PackTags[UnitNo.Shipping].Status.StateCurrent);

fbHmiHandShakeController(xEnable := TRUE,CylinderStatus := CylinderStatus,MotorStatus:=MotorStatus,FanucRobot := FanucRobot);

fbMachineHoming(
	xDone=> , 
	xBusy=> , 
	xError=> , 
	xExecute:= , 
	xAbort:= , 
	AllocateHome:= fbAllocateArea.fbAllocateHome, 
	StorageHome:= fbStorageArea.fbStorageHoming, 
	ShippingHome:= fbShippingArea.fbShippingHoming, 
	AllocateHomed:= fbAllocateArea.Homed, 
	StorageHomed:= fbStorageArea.Homed, 
	ShippingHomed:= fbShippingArea.Homed, 
	Homed:= MachineHomed, 
	TimeOut:= , 
	xAborted=> , 
	iErrorID=> , 
	ErrorMsg=> );
	
fbErrorHandler(
	xDone=> , 
	xBusy=> , 
	xError=> , 
	AlarmList:= PackTag.Admin.Alarm,
	AlarmHistory := PackTag.Admin.AlarmHistory, 
	HMI_AlarmMonitorList:= GVL_ADS.AlarmAllocation, 
	MaxRecords:= 1000, 
	ResetAllAlarms:= ,
	Reset := Machine_Reset OR tofResetDelay.Q , 
	EnableLogging:= , 
	ActiveAlarmCount=> , 
	TotalRecords=> , 
	SystemStatus=> );
	
fbBuzzCtrl(
	Execute:= GVL_ADS.BuzzCtrl.Command.Execute, 
	Abort:= GVL_ADS.BuzzCtrl.Command.Abort, 
	Reset:= GVL_ADS.BuzzCtrl.Command.Reset, 
	ObjectName:= , 
	Busy=> GVL_ADS.BuzzCtrl.Status.Busy, 
	Done=> GVL_ADS.BuzzCtrl.Status.Done, 
	Aborted=> , 
	Error=> GVL_ADS.BuzzCtrl.Status.Error, 
	ErrorID=> , 
	Status=> GVL_ADS.BuzzCtrl.Status.Status, 
	UniqueErrorCode=> , 
	Timer:=GVL_ADS.BuzzCtrl.BuzzTime, 
	Buzz=> BuzzCtrlUseBuzz);
	
fbMachineModeSwitch(
	Execute:= GVL_ADS.MachineMode.HandshakeBase.Execute,
	Abort:= ,
	Reset:= GVL_ADS.MachineMode.HandshakeBase.Reset,
	Pause:= ,
	ObjectName:= 'MachineModeSwitch',
	Busy=> GVL_ADS.MachineMode.HandshakeBase.Busy,
	Done=> GVL_ADS.MachineMode.HandshakeBase.Done,
	Aborted=> ,
	Error=> GVL_ADS.MachineMode.HandshakeBase.Error,
	ErrorID=> ,
	Status=> ,
	UniqueErrorCode=> ,
	ModeLink:= GVL_ADS.MachineMode,
	MachineCtrl_CurrentState := THIS^.eStateCurrent,
	MachineCtrl_CurrentMode := THIS^.eModeCommand,
	MachineHomed := MachineHomed);
	
fbBlink_05(ENABLE:= TRUE, TIMELOW:= T#0.25S, TIMEHIGH:= T#0.25S, OUT=> );
Allocate_EStopEdgeDetect(xInput := INPUT.bAllocate_EStopPb);
Storage_EstopEdgeDetect(xInput := INPUT.bStorage_EstopPb);

// HMi CameraBlow Ctrl
fbHmiCameraBlow(xInput := GVL_HMI.Storage.Manual.UpCV.CameraBlow);

TON_RobotReleaseResetCmd(IN:= RobotService_ResetCmd,PT:= T#500MS);
TON_RobotReleaseStartCmd(IN:= RobotService_StartCmd,PT:= T#500MS);
TON_Shipping_RobotRelease_ResetCmd(IN:= ShippingRobotService_ResetCmd,PT:= T#500MS);
TON_Shipping_RobotRelease_StartCmd(IN:= ShippingRobotService_StartCmd,PT:= T#500MS);
END_ACTION

ACTION A01_Cylinder:
cylinder.List.fbUpCV_FeedInPress1(xDone =>,
                                  xBusy =>,
                                  xError =>CylinderStatus.UpCV_FeedInPress1.Error,
                                  xEnable :=,
                                  FrontSensor :=,
                                  RearSensor :=,
                                  SetupPara := CurrentData.Cylinders.UpCV_FeedInPress1,
                                  CurrentCylinderType =>,
                                  InFrontPosition => CylinderStatus.UpCV_FeedInPress1.InFrontPosition,
                                  InRearPosition =>CylinderStatus.UpCV_FeedInPress1.InRearPosition,
                                  ExtendOutput => InternalOutput.bUpCV_FeedInPress1_Valve,
                                  RetractOutput =>);

cylinder.List.fbUpCV_FeedInPress2(xDone =>,
                                  xBusy =>,
                                  xError =>CylinderStatus.UpCV_FeedInPress2.Error,
                                  xEnable :=,
                                  FrontSensor :=,
                                  RearSensor :=,
                                  SetupPara := CurrentData.Cylinders.UpCV_FeedInPress2,
                                  CurrentCylinderType =>,
                                  InFrontPosition =>CylinderStatus.UpCV_FeedInPress2.InFrontPosition,
                                  InRearPosition =>CylinderStatus.UpCV_FeedInPress2.InRearPosition,
                                  ExtendOutput => InternalOutput.bUpCV_FeedInPress2_Valve,
                                  RetractOutput =>);

cylinder.List.fbUpCV_DiameterPress(xDone =>,
                                   xBusy =>,
                                   xError =>CylinderStatus.UpCV_DiameterPress.Error,
                                   xEnable :=,
                                   FrontSensor :=,
                                   RearSensor :=,
                                   SetupPara := CurrentData.Cylinders.UpCV_DiameterPress,
                                   CurrentCylinderType =>,
                                   InFrontPosition =>CylinderStatus.UpCV_DiameterPress.InFrontPosition,
                                   InRearPosition =>CylinderStatus.UpCV_DiameterPress.InRearPosition,
                                   ExtendOutput => InternalOutput.bUpCV_DiameterPress_Valve,
                                   RetractOutput =>);

cylinder.List.fbUpCV_CamaraPress1(xDone =>,
                                  xBusy =>,
                                  xError =>CylinderStatus.UpCV_CamaraPress1.Error,
                                  xEnable :=,
                                  FrontSensor :=,
                                  RearSensor :=,
                                  SetupPara := CurrentData.Cylinders.UpCV_CamaraPress1,
                                  CurrentCylinderType =>,
                                  InFrontPosition =>CylinderStatus.UpCV_CamaraPress1.InFrontPosition,
                                  InRearPosition =>CylinderStatus.UpCV_CamaraPress1.InRearPosition,
                                  ExtendOutput => InternalOutput.bUpCV_CamaraPress1_Valve,
                                  RetractOutput =>);

cylinder.List.fbUpCV_CamaraPress2(xDone =>,
                                  xBusy =>,
                                  xError =>CylinderStatus.UpCV_CamaraPress2.Error,
                                  xEnable :=,
                                  FrontSensor :=,
                                  RearSensor :=,
                                  SetupPara := CurrentData.Cylinders.UpCV_CamaraPress2,
                                  CurrentCylinderType =>,
                                  InFrontPosition =>CylinderStatus.UpCV_CamaraPress2.InFrontPosition,
                                  InRearPosition =>CylinderStatus.UpCV_CamaraPress2.InRearPosition,
                                  ExtendOutput => InternalOutput.bUpCV_CamaraPress2_Valve,
                                  RetractOutput =>);

cylinder.List.fbUpCV_CamaraPress3(xDone =>,
                                  xBusy =>,
                                  xError =>CylinderStatus.UpCV_CamaraPress3.Error,
                                  xEnable :=,
                                  FrontSensor :=,
                                  RearSensor :=,
                                  SetupPara := CurrentData.Cylinders.UpCV_CamaraPress3,
                                  CurrentCylinderType =>,
                                  InFrontPosition =>CylinderStatus.UpCV_CamaraPress3.InFrontPosition,
                                  InRearPosition =>CylinderStatus.UpCV_CamaraPress3.InRearPosition,
                                  ExtendOutput => InternalOutput.bUpCV_CamaraPress3_Valve,
                                  RetractOutput =>);

cylinder.List.fbUpCV_CamaraPress4(xDone =>, 
                                  xBusy =>,
                                  xError =>CylinderStatus.UpCV_CamaraPress4.Error,
                                  xEnable :=,
                                  FrontSensor :=,
                                  RearSensor :=,
                                  SetupPara := CurrentData.Cylinders.UpCV_CamaraPress4,
                                  CurrentCylinderType =>,
                                  InFrontPosition =>CylinderStatus.UpCV_CamaraPress4.InFrontPosition,
                                  InRearPosition =>CylinderStatus.UpCV_CamaraPress4.InRearPosition,
                                  ExtendOutput => InternalOutput.bUpCV_CamaraPress4_Valve,
                                  RetractOutput =>);

cylinder.List.fbUpCV_Block1(xDone =>,
                            xBusy =>,
                            xError =>CylinderStatus.UpCV_Block1.Error,
                            xEnable :=,
                            FrontSensor :=,
                            RearSensor := INPUT.bUpCV_Block1_RearSensor,
                            SetupPara := CurrentData.Cylinders.UpCV_Block1,
                            CurrentCylinderType =>,
                            InFrontPosition =>CylinderStatus.UpCV_Block1.InFrontPosition,
                            InRearPosition =>CylinderStatus.UpCV_Block1.InRearPosition,
                            ExtendOutput => InternalOutput.bUpCV_Block1_Up_Valve,
                            RetractOutput => InternalOutput.bUpCV_Block1_Down_Valve);
cylinder.List.fbUpCV_Block1.IsDoubleValve := TRUE;

cylinder.List.fbUpCV_Block2(xDone =>,
                            xBusy =>,
                            xError =>CylinderStatus.UpCV_Block2.Error,
                            xEnable :=,
                            FrontSensor :=,
                            RearSensor := INPUT.bUpCV_Block2_RearSensor,
                            SetupPara := CurrentData.Cylinders.UpCV_Block2,
                            CurrentCylinderType =>,
                            InFrontPosition =>CylinderStatus.UpCV_Block2.InFrontPosition,
                            InRearPosition =>CylinderStatus.UpCV_Block2.InRearPosition,
                            ExtendOutput => InternalOutput.bUpCV_Block2_Up_Valve,
                            RetractOutput => InternalOutput.bUpCV_Block2_Down_Valve);
cylinder.List.fbUpCV_Block2.IsDoubleValve := TRUE;

cylinder.List.fbUpCV_Block3(xDone =>,
                            xBusy =>,
                            xError =>CylinderStatus.UpCV_Block3.Error,
                            xEnable :=,
                            FrontSensor :=,
                            RearSensor := INPUT.bUpCV_Block3_RearSensor,
                            SetupPara := CurrentData.Cylinders.UpCV_Block3,
                            CurrentCylinderType =>,
                            InFrontPosition =>CylinderStatus.UpCV_Block3.InFrontPosition,
                            InRearPosition =>CylinderStatus.UpCV_Block3.InRearPosition,
                            ExtendOutput => InternalOutput.bUpCV_Block3_Up_Valve,
                            RetractOutput => InternalOutput.bUpCV_Block3_Down_Valve);
cylinder.List.fbUpCV_Block3.IsDoubleValve := TRUE;

cylinder.List.fbUpCV_DiameterHoriz(xDone =>,
                                   xBusy =>,
                                   xError =>CylinderStatus.UpCV_DiameterHoriz.Error,
                                   xEnable :=,
                                   FrontSensor := INPUT.bUpCV_DiameterHoriz_FrontSensor,
                                   RearSensor := INPUT.bUpCV_DiameterHoriz_RearSensor,
                                   SetupPara := CurrentData.Cylinders.UpCV_DiameterHoriz,
                                   CurrentCylinderType =>,
                                   InFrontPosition =>CylinderStatus.UpCV_DiameterHoriz.InFrontPosition,
                                   InRearPosition =>CylinderStatus.UpCV_DiameterHoriz.InRearPosition,
                                   ExtendOutput => InternalOutput.bUpCV_DiameterHoriz_Extend_Valve,
                                   RetractOutput => InternalOutput.bUpCV_DiameterHoriz_Retract_Valve);
cylinder.List.fbUpCV_DiameterHoriz.IsDoubleValve := TRUE;

cylinder.List.fbUpCV_DiameterVert(xDone =>,
                                  xBusy =>,
                                  xError =>CylinderStatus.UpCV_DiameterVert.Error,
                                  xEnable :=,
                                  FrontSensor := INPUT.bUpCV_DiameterVert_FrontSensor,
                                  RearSensor := INPUT.bUpCV_DiameterVert_RearSensor,
                                  SetupPara := CurrentData.Cylinders.UpCV_DiameterVert,
                                  CurrentCylinderType =>,
                                  InFrontPosition =>CylinderStatus.UpCV_DiameterVert.InFrontPosition,
                                  InRearPosition =>CylinderStatus.UpCV_DiameterVert.InRearPosition,
                                  ExtendOutput => InternalOutput.bUpCV_DiameterVert_Valve,
                                  RetractOutput =>);

cylinder.List.fbUpCV_DiameterClamp(xDone =>,
                                   xBusy =>,
                                   xError =>CylinderStatus.UpCV_DiameterClamp.Error,
                                   xEnable :=,
                                   FrontSensor :=,
                                   RearSensor :=,
                                   SetupPara := CurrentData.Cylinders.UpCV_DiameterClamp,
                                   CurrentCylinderType =>,
                                   InFrontPosition =>CylinderStatus.UpCV_DiameterClamp.InFrontPosition,
                                   InRearPosition =>CylinderStatus.UpCV_DiameterClamp.InRearPosition,
                                   ExtendOutput => InternalOutput.bUpCV_DiameterClamp_Close_Valve,
                                   RetractOutput => InternalOutput.bUpCV_DiameterClamp_Open_Valve);
cylinder.List.fbUpCV_DiameterClamp.IsDoubleValve := TRUE;

cylinder.List.fbStackPush(xDone =>,
                          xBusy =>,
                          xError =>CylinderStatus.StackPush.Error,
                          xEnable :=,
                          FrontSensor := INPUT.bStackPush_Pusher_FrontSensor,
                          RearSensor := INPUT.bStackPush_Pusher_RearSensor,
                          SetupPara := CurrentData.Cylinders.StackPush,
                          CurrentCylinderType =>,
                          InFrontPosition =>CylinderStatus.StackPush.InFrontPosition,
                          InRearPosition =>CylinderStatus.StackPush.InRearPosition,
                          ExtendOutput => InternalOutput.bStackPush_Valve,
                          RetractOutput =>);

cylinder.List.fbPullOutCV_AsidePress1(xDone =>,
                                      xBusy =>,
                                      xError =>CylinderStatus.PullOutCV_AsidePress1.Error,
                                      xEnable :=,
                                      FrontSensor :=,
                                      RearSensor :=,
                                      SetupPara := CurrentData.Cylinders.PullOutCV_AsidePress1,
                                      CurrentCylinderType =>,
                                      InFrontPosition =>CylinderStatus.PullOutCV_AsidePress1.InFrontPosition,
                                      InRearPosition =>CylinderStatus.PullOutCV_AsidePress1.InRearPosition,
                                      ExtendOutput => InternalOutput.bPullOutCV_AsidePress1_Valve,
                                      RetractOutput =>);

cylinder.List.fbPullOutCV_AsidePress2(xDone =>,
                                      xBusy =>,
                                      xError =>CylinderStatus.PullOutCV_AsidePress2.Error,
                                      xEnable :=,
                                      FrontSensor :=,
                                      RearSensor :=,
                                      SetupPara := CurrentData.Cylinders.PullOutCV_AsidePress2,
                                      CurrentCylinderType =>,
                                      InFrontPosition =>CylinderStatus.PullOutCV_AsidePress2.InFrontPosition,
                                      InRearPosition =>CylinderStatus.PullOutCV_AsidePress2.InRearPosition,
                                      ExtendOutput => InternalOutput.bPullOutCV_AsidePress2_Valve,
                                      RetractOutput =>);

cylinder.List.fbPullOutCV_AsideBlock(xDone =>,
                                     xBusy =>,
                                     xError =>CylinderStatus.PullOutCV_AsideBlock.Error,
                                     xEnable :=,
                                     FrontSensor :=,
                                     RearSensor := INPUT.bPullOutCV_AsideBlock_RearSensor,
                                     SetupPara := CurrentData.Cylinders.PullOutCV_AsideBlock,
                                     CurrentCylinderType =>,
                                     InFrontPosition =>CylinderStatus.PullOutCV_AsideBlock.InFrontPosition,
                                     InRearPosition =>CylinderStatus.PullOutCV_AsideBlock.InRearPosition,
                                     ExtendOutput => InternalOutput.bPullOutCV_AsideBlock_Valve,
                                     RetractOutput =>);

cylinder.List.fbPullOutCV_BsidePress1(xDone =>,
                                      xBusy =>,
                                      xError =>CylinderStatus.PullOutCV_BsidePress1.Error,
                                      xEnable :=,
                                      FrontSensor :=,
                                      RearSensor :=,
                                      SetupPara := CurrentData.Cylinders.PullOutCV_BsidePress1,
                                      CurrentCylinderType =>,
                                      InFrontPosition =>CylinderStatus.PullOutCV_BsidePress1.InFrontPosition,
                                      InRearPosition =>CylinderStatus.PullOutCV_BsidePress1.InRearPosition,
                                      ExtendOutput => InternalOutput.bPullOutCV_BsidePress1_Valve,
                                      RetractOutput =>);

cylinder.List.fbPullOutCV_BsidePress2(xDone =>,
                                      xBusy =>,
                                      xError =>CylinderStatus.PullOutCV_BsidePress2.Error,
                                      xEnable :=,
                                      FrontSensor :=,
                                      RearSensor :=,
                                      SetupPara := CurrentData.Cylinders.PullOutCV_BsidePress2,
                                      CurrentCylinderType =>,
                                      InFrontPosition =>CylinderStatus.PullOutCV_BsidePress2.InFrontPosition,
                                      InRearPosition =>CylinderStatus.PullOutCV_BsidePress2.InRearPosition,
                                      ExtendOutput => InternalOutput.bPullOutCV_BsidePress2_Valve,
                                      RetractOutput =>);

cylinder.List.fbPullOutCV_BsideBlock(xDone =>,
                                     xBusy =>,
                                     xError =>CylinderStatus.PullOutCV_BsideBlock.Error,
                                     xEnable :=,
                                     FrontSensor :=,
                                     RearSensor := INPUT.bPullOutCV_BsideBlock_RearSensor,
                                     SetupPara := CurrentData.Cylinders.PullOutCV_BsideBlock,
                                     CurrentCylinderType =>,
                                     InFrontPosition =>CylinderStatus.PullOutCV_BsideBlock.InFrontPosition,
                                     InRearPosition =>CylinderStatus.PullOutCV_BsideBlock.InRearPosition,
                                     ExtendOutput => InternalOutput.bPullOutCV_BsideBlock_Valve,
                                     RetractOutput =>);

cylinder.List.fbLowCV_Press1(xDone =>,
                             xBusy =>,
                             xError =>CylinderStatus.LowCV_Press1.Error,
                             xEnable :=,
                             FrontSensor :=,
                             RearSensor :=,
                             SetupPara := CurrentData.Cylinders.LowCV_Press1,
                             CurrentCylinderType =>,
                             InFrontPosition =>CylinderStatus.LowCV_Press1.InFrontPosition,
                             InRearPosition =>CylinderStatus.LowCV_Press1.InRearPosition,
                             ExtendOutput => InternalOutput.bLowCV_Press1_Valve,
                             RetractOutput =>);

cylinder.List.fbLowCV_Press2(xDone =>,
                             xBusy =>,
                             xError =>CylinderStatus.LowCV_Press2.Error,
                             xEnable :=,
                             FrontSensor :=,
                             RearSensor :=,
                             SetupPara := CurrentData.Cylinders.LowCV_Press2,
                             CurrentCylinderType =>,
                             InFrontPosition =>CylinderStatus.LowCV_Press2.InFrontPosition,
                             InRearPosition =>CylinderStatus.LowCV_Press2.InRearPosition,
                             ExtendOutput => InternalOutput.bLowCV_Press2_Valve,
                             RetractOutput =>);

cylinder.List.fbLowCV_Press3(xDone =>,
                             xBusy =>,
                             xError =>CylinderStatus.LowCV_Press3.Error,
                             xEnable :=,
                             FrontSensor :=,
                             RearSensor :=,
                             SetupPara := CurrentData.Cylinders.LowCV_Press3,
                             CurrentCylinderType =>,
                             InFrontPosition =>CylinderStatus.LowCV_Press3.InFrontPosition,
                             InRearPosition =>CylinderStatus.LowCV_Press3.InRearPosition,
                             ExtendOutput => InternalOutput.bLowCV_Press3_Valve,
                             RetractOutput =>);

cylinder.List.fbLowCV_Press4(xDone =>,
                             xBusy =>,
                             xError =>CylinderStatus.LowCV_Press4.Error,
                             xEnable :=,
                             FrontSensor :=,
                             RearSensor :=,
                             SetupPara := CurrentData.Cylinders.LowCV_Press4,
                             CurrentCylinderType =>,
                             InFrontPosition =>CylinderStatus.LowCV_Press4.InFrontPosition,
                             InRearPosition =>CylinderStatus.LowCV_Press4.InRearPosition,
                             ExtendOutput => InternalOutput.bLowCV_Press4_Valve,
                             RetractOutput =>);

cylinder.List.fbLowCV_Block1(xDone =>,
                             xBusy =>,
                             xError =>CylinderStatus.LowCV_Block1.Error,
                             xEnable :=,
                             FrontSensor :=,
                             RearSensor := INPUT.bLowCV_Block1_RearSensor,
                             SetupPara := CurrentData.Cylinders.LowCV_Block1,
                             CurrentCylinderType =>,
                             InFrontPosition =>CylinderStatus.LowCV_Block1.InFrontPosition,
                             InRearPosition =>CylinderStatus.LowCV_Block1.InRearPosition,
                             ExtendOutput => InternalOutput.bLowCV_Block1_Down_Valve,
                             RetractOutput => InternalOutput.bLowCV_Block1_Up_Valve);
cylinder.List.fbLowCV_Block1.IsDoubleValve := TRUE;

cylinder.List.fbLowCV_Block2(xDone =>,
                             xBusy =>,
                             xError =>CylinderStatus.LowCV_Block2.Error,
                             xEnable :=,
                             FrontSensor :=,
                             RearSensor := INPUT.bLowCV_Block2_RearSensor,
                             SetupPara := CurrentData.Cylinders.LowCV_Block2,
                             CurrentCylinderType =>,
                             InFrontPosition =>CylinderStatus.LowCV_Block2.InFrontPosition,
                             InRearPosition =>CylinderStatus.LowCV_Block2.InRearPosition,
                             ExtendOutput => InternalOutput.bLowCV_Block2_Down_Valve,
                             RetractOutput => InternalOutput.bLowCV_Block2_Up_Valve);
cylinder.List.fbLowCV_Block2.IsDoubleValve := TRUE;

cylinder.List.fbAllocateRobot_LeftVert1(xDone =>,
                                        xBusy =>,
                                        xError =>CylinderStatus.AllocateRobot_LeftVert1.Error,
                                        xEnable :=,
                                        FrontSensor := INPUT.bAllocateRobot_LeftVert1_LowSensor,
                                        RearSensor := INPUT.bAllocateRobot_LeftVert1_HighSensor,
                                        SetupPara := CurrentData.Cylinders.AllocateRobot_LeftVert1,
                                        CurrentCylinderType =>,
                                        InFrontPosition =>CylinderStatus.AllocateRobot_LeftVert1.InFrontPosition,
                                        InRearPosition =>CylinderStatus.AllocateRobot_LeftVert1.InRearPosition,
                                        ExtendOutput => InternalOutput.bAllocateRobot_LeftVert1_Valve,
                                        RetractOutput =>);

cylinder.List.fbAllocateRobot_LeftVert2(xDone =>,
                                        xBusy =>,
                                        xError =>CylinderStatus.AllocateRobot_LeftVert2.Error,
                                        xEnable :=,
                                        FrontSensor := input.bAllocateRobot_LeftVert2_LowSensor,
                                        RearSensor := input.bAllocateRobot_LeftVert2_HighSensor,
                                        SetupPara := CurrentData.Cylinders.AllocateRobot_LeftVert2,
                                        CurrentCylinderType =>,
                                        InFrontPosition =>CylinderStatus.AllocateRobot_LeftVert2.InFrontPosition,
                                        InRearPosition =>CylinderStatus.AllocateRobot_LeftVert2.InRearPosition,
                                        ExtendOutput => InternalOutput.bAllocateRobot_LeftVert2_Valve,
                                        RetractOutput =>);

cylinder.List.fbAllocateRobot_RightVert1(xDone =>,
                                         xBusy =>,
                                         xError =>CylinderStatus.AllocateRobot_RightVert1.Error,
                                         xEnable :=,
                                         FrontSensor := input.bAllocateRobot_RightVert1_LowSensor,
                                         RearSensor := input.bAllocateRobot_RightVert1_HighSensor,
                                         SetupPara := CurrentData.Cylinders.AllocateRobot_RightVert1,
                                         CurrentCylinderType =>,
                                         InFrontPosition =>CylinderStatus.AllocateRobot_RightVert1.InFrontPosition,
                                         InRearPosition =>CylinderStatus.AllocateRobot_RightVert1.InRearPosition,
                                         ExtendOutput => InternalOutput.bAllocateRobot_RightVert1_Valve,
                                         RetractOutput =>);

cylinder.List.fbAllocateRobot_RightVert2(xDone =>,
                                         xBusy =>,
                                         xError =>CylinderStatus.AllocateRobot_RightVert2.Error,
                                         xEnable :=,
                                         FrontSensor := input.bAllocateRobot_RightVert2_LowSensor,
                                         RearSensor := input.bAllocateRobot_RightVert2_HighSensor,
                                         SetupPara := CurrentData.Cylinders.AllocateRobot_RightVert2,
                                         CurrentCylinderType =>,
                                         InFrontPosition =>CylinderStatus.AllocateRobot_RightVert2.InFrontPosition,
                                         InRearPosition =>CylinderStatus.AllocateRobot_RightVert2.InRearPosition,
                                         ExtendOutput => InternalOutput.bAllocateRobot_RightVert2_Valve,
                                         RetractOutput =>);

